(* CODESYS project SPT_XTS.library
   Version: 4.0.0
   Title: SPT XTS
   DefaultNamespace: SPT_XTS
   Placeholder: SPT XTS
   Company: Beckhoff Automation LLC

Project tree, tasks and I/O mapping:
  libraries: SPT Base Types, * (Beckhoff Automation LLC); SPT Event Logger, * (Beckhoff Automation LLC); SPT Utilities, * (Beckhoff Automation LLC); Tc2_Math, * (Beckhoff Automation GmbH); Tc2_MC2, * (Beckhoff Automation GmbH); Tc2_Standard, * (Beckhoff Automation GmbH); Tc2_System, * (Beckhoff Automation GmbH); Tc2_Utilities, * (Beckhoff Automation GmbH); Tc3_EventLogger, * (Beckhoff Automation GmbH); Tc3_JsonXml, * (Beckhoff Automation GmbH); Tc3_McCollisionAvoidance, * (Beckhoff Automation GmbH); Tc3_McCoordinatedMotion, * (Beckhoff Automation GmbH); Tc3_Module, * (Beckhoff Automation GmbH); Tc3_XTS_Utility, * (Beckhoff Automation GmbH); Tc3_PackML_V3, * (Beckhoff Automation GmbH)
  Application Station Reference/
    DUTs/
      data type E_ApplicationStationState
    function block FB_XTS_QueueStation [ST]: CanAcceptMover, CanReleaseMover, Resetting, Execute, GetMovers, MaxNumberOfMovers
    function block FB_XTS_SimpleStation [ST]: Execute, SimulatedProcessTime
  GVLs/
    global variables CONSTANTS
    global variables XTS
  Movers/
    data type E_InitializeState_Mover
    function block FB_XTS_Mover [ST]: CyclicLogic, Disable, Enable, GearInPosCA, JoinGroup, LeaveGroup, MoveAbsoluteCA, MoveRelativeCA, Reset, Stop, Acceleration, Deceleration, Gap, Jerk, Velocity, ActualAcceleration, ActualPosition, ActualPositionModulo, ActualTorque, ActualVelocity, PositionLag, SetAcceleration, SetPosition, SetPositionModulo, SetVelocity, Enabled, InPosition, InSync, Stopped, Axis, IsMoverInPosition, LimitBipolarCurrent, MoverID, Override, Station, Trace, TraceMoveCommand, TraceWriteBoolParameter, TraceWriteParameter, AxisRefLinked, CurrentPart, CurrentPartOID, CurrentTrack, CurrentTrackOID, FB_reinit, Group, Initialize
    interface I_XTS_Mover: Disable, Enable, GearInPosCA, JoinGroup, LeaveGroup, MoveAbsoluteCA, MoveRelativeCA, Reset, Stop, Acceleration, Deceleration, Jerk, Velocity, ActualAcceleration, ActualPosition, ActualPositionModulo, ActualTorque, ActualVelocity, PositionLag, SetAcceleration, SetPosition, SetPositionModulo, SetVelocity, Enabled, InPosition, InSync, Stopped, Axis, IsMoverInPosition, LimitBipolarCurrent, MoverID, Override, Station
    data type ST_GearInPosCAParameters
    data type ST_MoveDynamics
  Parts/
    data type E_InitializeState_Part
    function block FB_XTS_Part [ST]: CyclicLogic, Initialize, ModuleCoEData, Name, ReadyToEnable, Reset
    interface I_XTS_Part: Name, ReadyToEnable
  Project Information/
    function F_GetCompany [ST]
    function F_GetTitle [ST]
    function F_GetVersion [ST]
  Stations/
    data type E_Colors_ARGB
    data type E_InitializeState_Station
    function block FB_XTS_InfoStation [ST]: CyclicLogic, ApplicationStation, Color, GetMover, GetStopPositionOnTrack, MoverQueue, NumberOfStops, StopPositions, GiveMover, StationName, TakeMover, Initialize, IsAQueue, MoverIDsAssigned, ReleaseAllMovers, StationID
    function block FB_XTS_StationBase [ST]: CanAcceptMover, CanReleaseMover, Config, InfoStation, TrackOID, Resetting, Stopping, HMIPermissions, Initialize, GetMovers, GetStopPosition, CyclicLogic, NumberOfAssignedMovers, NumberOfStops, StopPositions
    interface I_XTS_ApplicationStation: CanAcceptMover, CanReleaseMover, Config, InfoStation, Name, TrackOID
    interface I_XTS_InfoStation: ApplicationStation, Color, GetMover, GetStopPositionOnTrack, MoverQueue, NumberOfStops, StopPositions
    interface I_XTS_StationNeighbor: GiveMover, StationName, TakeMover
    data type ST_XTSStationConfig
  Tracks/
    data type E_InitializeState_Track
    function block FB_XTS_Track [ST]: CyclicLogic, GetTrackPositionByPart, IsClosed, Length, Name, Initialize
    interface I_XTS_Track: GetTrackPositionByPart, IsClosed, Length, Name
  Utilities/
    function block FB_MoverQueue [ST]: Clear, Count, Dequeue, Enqueue, FirstMover, LastMover, MoverIDs, Queue
    function block FB_RingBuffer_MCGearInPosCA [ST]: CurrentFB, GetNewFB
    function block FB_RingBuffer_MCMoveAbsoluteCA [ST]: CurrentFB, GetNewFB
    function block FB_RingBuffer_MCMoveRelativeCA [ST]: CurrentFB, GetNewFB
    function block FB_TrackingRegister_Movers [ST]: Check, Clear, NumberCompleted, Reset, Set
    function block FB_TrackingRegister_Stations [ST]: Check, Clear, Complete, NumberCompleted, Reset, Set, StationsToTrack
  Version/
    global variables Global_Version
  XPU/
    DUTs/
      data type E_MoverAssignmentRecoverySource
      data type E_XPUColdStartRecoveryState
      data type E_XPUInitializeState
      data type E_XPUInitializeState_CAGroups
      data type E_XPUInitializeState_Environment
      data type E_XPUInitializeState_InfoStations
      data type E_XPUInitializeState_XPU
      data type E_XTSState
      data type ST_MoverAssignmentData
      data type ST_StationNeighbors
    function block FB_Component_XPU [ST]: CyclicLogic, GetPositionOnTrack, GiveMover, InSimulationMode, CreateEvents, Monitoring, Initialize_CAGroups, Initialize_Environment, Initialize_InfoStations, Initialize_XPU, Initialize, ClearAllEvents, CollectRecoveryData, FindRecoveryCandidates, MoverAssignmentRecovery, ReassignMovers, RestoreBackupData, SetError, SetStationNeighbors, SortMoverBuckets, Trace, ClearMoverAssignments, Disable, Enable, FB_init, MoverAssignmentStorageLocation, PartCoEData, Reset, State, Stations
    interface I_XTS_Xpu: GetPositionOnTrack, GiveMover, InSimulationMode
  00000000-0000-0000-0000-000000000000|LICENSE
  LICENSE
  global variables Parameters_XTS
*)

// Application Station Reference/DUTs/E_ApplicationStationState
{attribute 'qualified_only'}
{attribute 'strict'}
TYPE E_ApplicationStationState : (
		eApplicationStationState_Init		   := 0,
		eApplicationStationState_GetMovers	   := 1,
		eApplicationStationState_InProcess	   := 2,
		eApplicationStationState_ReleaseMovers := 4
	) DWORD;
END_TYPE

// Movers/E_InitializeState_Mover
{attribute 'qualified_only'}
{attribute 'strict'}
TYPE E_InitializeState_Mover : (
		eInitializeStateMover_Check,
		eInitializeStateMover_GetSoftDriveInterfaces,
		eInitializeStateMover_GetSoftDriveInterfaces_Encoder,
		eInitializeStateMover_GetSoftDriveInterfaces_FeedForward,
		eInitializeStateMover_GetSoftDriveInterfaces_Filters,
		eInitializeStateMover_GetSoftDriveInterfaces_Interpolator,
		eInitializeStateMover_GetSoftDriveInterfaces_PositionController,
		eInitializeStateMover_GetSoftDriveInterfaces_VelocityController,
		eInitializeStateMover_ReadTcIOParameters,
		eInitializeStateMover_CheckDriveLinks,
		eInitializeStateMover_ReadNCParameters,
		eInitializeStateMover_Complete,
		eInitializeStateMover_Failed
	);
END_TYPE

// Movers/ST_GearInPosCAParameters
TYPE ST_GearInPosCAParameters :
	STRUCT
		RatioNumerator		: MC_LREAL		   := 1;
		RatioDenumerator	: UINT			   := 1;
		MasterSyncPosition	: MC_LREAL		   := MC_INVALID;
		SlaveSyncPosition	: MC_LREAL		   := MC_INVALID;
		SyncStrategy		: MC_SYNC_STRATEGY := MC_SYNC_STRATEGY.mcSyncStrategyEarly;
		SyncMode			: MC_SYNC_MODE	   := MC_SYNC_MODE.mcSyncModePositive;
		MasterStartDistance : MC_LREAL		   := MC_IGNORE;
		Velocity			: MC_LREAL		   := MC_INVALID;
		Acceleration		: MC_LREAL		   := MC_DEFAULT;
		Deceleration		: MC_LREAL		   := MC_DEFAULT;
		Jerk				: MC_LREAL		   := MC_DEFAULT;
		Gap					: MC_LREAL		   := MC_DEFAULT;
		BufferMode			: MC_BUFFER_MODE   := mcAborting;
		Options				: ST_GearInPosCAOptions;
	END_STRUCT
END_TYPE

// Movers/ST_MoveDynamics
TYPE ST_MoveDynamics :
	STRUCT
		Velocity	 : LREAL := 200;
		Acceleration : LREAL := MC_DEFAULT;
		Deceleration : LREAL := MC_DEFAULT;
		Jerk		 : LREAL := MC_DEFAULT;
	END_STRUCT
END_TYPE

// Parts/E_InitializeState_Part
{attribute 'qualified_only'}
{attribute 'strict'}
TYPE E_InitializeState_Part : (
		eInitializeStatePart_Check,
		eInitializeStatePart_GetModuleInterfaces,
		eInitializeStatePart_GetControlAreaInterfaces,
		eInitializeStatePart_Complete,
		eInitializeStatePart_Failed
	);
END_TYPE

// Stations/E_Colors_ARGB
{attribute 'qualified_only'}
TYPE E_Colors_ARGB : (
		Darkred				 := 16#FF8B0000, //	rgb(139,0,0)
		Brown				 := 16#FFA52A2A, //	rgb(165,42,42)
		Firebrick			 := 16#FFB22222, //	rgb(178,34,34)
		Crimson				 := 16#FFDC143C, //	rgb(220,20,60)
		Red					 := 16#FFFF0000, //	rgb(255,0,0)
		Tomato				 := 16#FFFF6347, //	rgb(255,99,71)
		Coral				 := 16#FFFF7F50, //	rgb(255,127,80)
		Indianred			 := 16#FFCD5C5C, //	rgb(205,92,92)
		Lightcoral			 := 16#FFF08080, //	rgb(240,128,128)
		Darksalmon			 := 16#FFE9967A, //	rgb(233,150,122)
		Salmon				 := 16#FFFA8072, //	rgb(250,128,114)
		Lightsalmon			 := 16#FFFFA07A, //	rgb(255,160,122)
		Orangered			 := 16#FFFF4500, //	rgb(255,69,0)
		Darkorange			 := 16#FFFF8C00, //	rgb(255,140,0)
		Orange				 := 16#FFFFA500, //	rgb(255,165,0)
		Gold				 := 16#FFFFD700, //	rgb(255,215,0)
		Darkgoldenrod		 := 16#FFB8860B, //	rgb(184,134,11)
		Goldenrod			 := 16#FFDAA520, //	rgb(218,165,32)
		Palegoldenrod		 := 16#FFEEE8AA, //	rgb(238,232,170)
		Darkkhaki			 := 16#FFBDB76B, //	rgb(189,183,107)
		Khaki				 := 16#FFF0E68C, //	rgb(240,230,140)
		Olive				 := 16#FF808000, //	rgb(128,128,0)
		Yellow				 := 16#FFFFFF00, //	rgb(255,255,0)
		Yellowgreen			 := 16#FF9ACD32, //	rgb(154,205,50)
		Darkolivegreen		 := 16#FF556B2F, //	rgb(85,107,47)
		Olivedrab			 := 16#FF6B8E23, //	rgb(107,142,35)
		Lawngreen			 := 16#FF7CFC00, //	rgb(124,252,0)
		Chartreuse			 := 16#FF7FFF00, //	rgb(127,255,0)
		Greenyellow			 := 16#FFADFF2F, //	rgb(173,255,47)
		Darkgreen			 := 16#FF006400, //	rgb(0,100,0)
		Green				 := 16#FF008000, //	rgb(0,128,0)
		Forestgreen			 := 16#FF228B22, //	rgb(34,139,34)
		Lime				 := 16#FF00FF00, //	rgb(0,255,0)
		Limegreen			 := 16#FF32CD32, //	rgb(50,205,50)
		Lightgreen			 := 16#FF90EE90, //	rgb(144,238,144)
		Palegreen			 := 16#FF98FB98, //	rgb(152,251,152)
		Darkseagreen		 := 16#FF8FBC8F, //	rgb(143,188,143)
		Mediumspringgreen	 := 16#FF00FA9A, //	rgb(0,250,154)
		Springgreen			 := 16#FF00FF7F, //	rgb(0,255,127)
		Seagreen			 := 16#FF2E8B57, //	rgb(46,139,87)
		Mediumaquamarine	 := 16#FF66CDAA, //	rgb(102,205,170)
		Mediumseagreen		 := 16#FF3CB371, //	rgb(60,179,113)
		Lightseagreen		 := 16#FF20B2AA, //	rgb(32,178,170)
		Darkslategray		 := 16#FF2F4F4F, //	rgb(47,79,79)
		Teal				 := 16#FF008080, //	rgb(0,128,128)
		Darkcyan			 := 16#FF008B8B, //	rgb(0,139,139)
		Aqua				 := 16#FF00FFFF, //	rgb(0,255,255)
		Lightcyan			 := 16#FFE0FFFF, //	rgb(224,255,255)
		Darkturquoise		 := 16#FF00CED1, //	rgb(0,206,209)
		Turquoise			 := 16#FF40E0D0, //	rgb(64,224,208)
		Mediumturquoise		 := 16#FF48D1CC, //	rgb(72,209,204)
		Paleturquoise		 := 16#FFAFEEEE, //	rgb(175,238,238)
		Aquamarine			 := 16#FF7FFFD4, //	rgb(127,255,212)
		Powderblue			 := 16#FFB0E0E6, //	rgb(176,224,230)
		Cadetblue			 := 16#FF5F9EA0, //	rgb(95,158,160)
		Steelblue			 := 16#FF4682B4, //	rgb(70,130,180)
		Cornflowerblue		 := 16#FF6495ED, //	rgb(100,149,237)
		Deepskyblue			 := 16#FF00BFFF, //	rgb(0,191,255)
		Dodgerblue			 := 16#FF1E90FF, //	rgb(30,144,255)
		Lightblue			 := 16#FFADD8E6, //	rgb(173,216,230)
		Skyblue				 := 16#FF87CEEB, //	rgb(135,206,235)
		Lightskyblue		 := 16#FF87CEFA, //	rgb(135,206,250)
		Midnightblue		 := 16#FF191970, //	rgb(25,25,112)
		Navy				 := 16#FF000080, //	rgb(0,0,128)
		Darkblue			 := 16#FF00008B, //	rgb(0,0,139)
		Mediumblue			 := 16#FF0000CD, //	rgb(0,0,205)
		Blue				 := 16#FF0000FF, //	rgb(0,0,255)
		Royalblue			 := 16#FF4169E1, //	rgb(65,105,225)
		Blueviolet			 := 16#FF8A2BE2, //	rgb(138,43,226)
		Indigo				 := 16#FF4B0082, //	rgb(75,0,130)
		Darkslateblue		 := 16#FF483D8B, //	rgb(72,61,139)
		Slateblue			 := 16#FF6A5ACD, //	rgb(106,90,205)
		Mediumslateblue		 := 16#FF7B68EE, //	rgb(123,104,238)
		Mediumpurple		 := 16#FF9370DB, //	rgb(147,112,219)
		Darkmagenta			 := 16#FF8B008B, //	rgb(139,0,139)
		Darkviolet			 := 16#FF9400D3, //	rgb(148,0,211)
		Darkorchid			 := 16#FF9932CC, //	rgb(153,50,204)
		Mediumorchid		 := 16#FFBA55D3, //	rgb(186,85,211)
		Purple				 := 16#FF800080, //	rgb(128,0,128)
		Thistle				 := 16#FFD8BFD8, //	rgb(216,191,216)
		Plum				 := 16#FFDDA0DD, //	rgb(221,160,221)
		Violet				 := 16#FFEE82EE, //	rgb(238,130,238)
		Magenta				 := 16#FFFF00FF, //	rgb(255,0,255)
		Orchid				 := 16#FFDA70D6, //	rgb(218,112,214)
		Mediumvioletred		 := 16#FFC71585, //	rgb(199,21,133)
		Palevioletred		 := 16#FFDB7093, //	rgb(219,112,147)
		Deeppink			 := 16#FFFF1493, //	rgb(255,20,147)
		Hotpink				 := 16#FFFF69B4, //	rgb(255,105,180)
		Lightpink			 := 16#FFFFB6C1, //	rgb(255,182,193)
		Pink				 := 16#FFFFC0CB, //	rgb(255,192,203)
		Antiquewhite		 := 16#FFFAEBD7, //	rgb(250,235,215)
		Beige				 := 16#FFF5F5DC, //	rgb(245,245,220)
		Bisque				 := 16#FFFFE4C4, //	rgb(255,228,196)
		Blanchedalmond		 := 16#FFFFEBCD, //	rgb(255,235,205)
		Wheat				 := 16#FFF5DEB3, //	rgb(245,222,179)
		Cornsilk			 := 16#FFFFF8DC, //	rgb(255,248,220)
		Lemonchiffon		 := 16#FFFFFACD, //	rgb(255,250,205)
		LightGoldenRodYellow := 16#FFFAFAD2, //	rgb(250,250,210)
		LightYellow			 := 16#FFFFFFE0, //	rgb(255,255,224)
		SaddleBrown			 := 16#FF8B4513, //	rgb(139,69,19)
		Sienna				 := 16#FFA0522D, //	rgb(160,82,45)
		Chocolate			 := 16#FFD2691E, //	rgb(210,105,30)
		Peru				 := 16#FFCD853F, //	rgb(205,133,63)
		SandyBrown			 := 16#FFF4A460, //	rgb(244,164,96)
		BurlyWood			 := 16#FFDEB887, //	rgb(222,184,135)
		RosyBrown			 := 16#FFBC8F8F, //	rgb(188,143,143)
		Moccasin			 := 16#FFFFE4B5, //	rgb(255,228,181)
		NavajoWhite			 := 16#FFFFDEAD, //	rgb(255,222,173)
		PeachPuff			 := 16#FFFFDAB9, //	rgb(255,218,185)
		MistyRose			 := 16#FFFFE4E1, //	rgb(255,228,225)
		LavenderBlush		 := 16#FFFFF0F5, //	rgb(255,240,245)
		Linen				 := 16#FFFAF0E6, //	rgb(250,240,230)
		OldLace				 := 16#FFFDF5E6, //	rgb(253,245,230)
		PapayaWhip			 := 16#FFFFEFD5, //	rgb(255,239,213)
		Seashell			 := 16#FFFFF5EE, //	rgb(255,245,238)
		MintCream			 := 16#FFF5FFFA, //	rgb(245,255,250)
		SlateGray			 := 16#FF708090, //	rgb(112,128,144)
		LightSlateGray		 := 16#FF778899, //	rgb(119,136,153)
		LightSteelBlue		 := 16#FFB0C4DE, //	rgb(176,196,222)
		Lavender			 := 16#FFE6E6FA, //	rgb(230,230,250)
		FloralWhite			 := 16#FFFFFAF0, //	rgb(255,250,240)
		AliceBlue			 := 16#FFF0F8FF, //	rgb(240,248,255)
		GhostWhite			 := 16#FFF8F8FF, //	rgb(248,248,255)
		HoneyDew			 := 16#FFF0FFF0, //	rgb(240,255,240)
		Ivory				 := 16#FFFFFFF0, //	rgb(255,255,240)
		Azure				 := 16#FFF0FFFF, //	rgb(240,255,255)
		Snow				 := 16#FFFFFAFA, //	rgb(255,250,250)
		Black				 := 16#FF000000, //	rgb(0,0,0)
		DimGray				 := 16#FF696969, //	rgb(105,105,105)
		Gray				 := 16#FF808080, //	rgb(128,128,128)
		DarkGray			 := 16#FFA9A9A9, //	rgb(169,169,169)
		Silver				 := 16#FFC0C0C0, //	rgb(192,192,192)
		LightGray			 := 16#FFD3D3D3, //	rgb(211,211,211)
		Gainsboro			 := 16#FFDCDCDC, //	rgb(220,220,220)
		WhiteSmoke			 := 16#FFF5F5F5, //	rgb(245,245,245)
		White				 := 16#FFFFFFFF	 //	rgb(255,255,255)
	) UDINT;
END_TYPE

// Stations/E_InitializeState_Station
{attribute 'qualified_only'}
{attribute 'strict'}
TYPE E_InitializeState_Station : (
		eInitializeStateStation_Check,
		eInitializeStateStation_GetPartInfo,
		eInitializeStateStation_GetStopPositions,
		eInitializeStateStation_Complete,
		eInitializeStateStation_Failed
	);
END_TYPE

// Stations/ST_XTSStationConfig
TYPE ST_XTSStationConfig :
	STRUCT
		IsAQueueStation : BOOL; // Can accept movers on cold start recovery (station limits will be ignored!!)
		OverrideGap		: BOOL;
		Gap				: LREAL;
		Dynamics		: ST_MoveDynamics;
	END_STRUCT
END_TYPE

// Tracks/E_InitializeState_Track
{attribute 'qualified_only'}
{attribute 'strict'}
TYPE E_InitializeState_Track : (
		eInitializeStateTrack_Check,
		eInitializeStateTrack_GetPartInfo,
		eInitializeStateTrack_Complete,
		eInitializeStateTrack_Failed
	);
END_TYPE

// XPU/DUTs/E_MoverAssignmentRecoverySource
{attribute 'qualified_only'}
{attribute 'strict'}
TYPE E_MoverAssignmentRecoverySource : (
		eMoverAssignmentRecoverySource_NoBackup	  := 0,
		eMoverAssignmentRecoverySource_NOVRAM	  := 1,
		eMoverAssignmentRecoverySource_Persistent := 2
	);
END_TYPE

// XPU/DUTs/E_XPUColdStartRecoveryState
{attribute 'qualified_only'}
{attribute 'strict'}
TYPE E_XPUColdStartRecoveryState : (
		eXPUColdStartRecoveryState_CheckMover1Config := 0,
		eXPUColdStartRecoveryState_WaitForDriveReady,
		eXPUColdStartRecoveryState_StartMover1Detection,
		eXPUColdStartRecoveryState_WaitForMover1DetectionComplete,
		eXPUColdStartRecoveryState_CheckPersistentDataSource,
		eXPUColdStartRecoveryState_RestorePersistentStationMoverAssignments,
		eXPUColdStartRecoveryState_RestoreNOVRAMStationMoverAssignments,
		eXPUColdStartRecoveryState_LookForRecoveryCandidates,
		eXPUColdStartRecoveryState_ForceMoversOntoCandidates,
		eXPUColdStartRecoveryState_RecoveryComplete
	);
END_TYPE

// XPU/DUTs/E_XPUInitializeState
{attribute 'qualified_only'}
{attribute 'strict'}
TYPE E_XPUInitializeState : (
		eXPUInitializeState_Environment,
		eXPUInitializeState_CAGroups,
		eXPUInitializeState_XPU,
		eXPUInitializeState_InfoStations,
		eXPUInitializeState_Parts,
		eXPUInitializeState_Tracks,
		eXPUInitializeState_Movers,
		eXPUInitializeState_Stations,
		eXPUInitializeState_AttemptMoverRecovery,
		eXPUInitializeState_Complete,
		eXPUInitializeState_Failed
	);
END_TYPE

// XPU/DUTs/E_XPUInitializeState_CAGroups
{attribute 'qualified_only'}
{attribute 'strict'}
TYPE E_XPUInitializeState_CAGroups : (
		eXPUInitializeStateCAGroups_CheckMapping,
		eXPUInitializeStateCAGroups_FindGroupID,
		eXPUInitializeStateCAGroups_CheckGroupInitialized,
		eXPUInitializeStateCAGroups_Complete,
		eXPUInitializeStateCAGroups_Failed
	);
END_TYPE

// XPU/DUTs/E_XPUInitializeState_Environment
{attribute 'qualified_only'}
{attribute 'strict'}
TYPE E_XPUInitializeState_Environment : (
		eXPUInitializeStateEnvironment_Check,
		eXPUInitializeStateEnvironment_InitializeEnvironment,
		eXPUInitializeStateEnvironment_GetXPUCount,
		eXPUInitializeStateEnvironment_GetXPUOIDs,
		eXPUInitializeStateEnvironment_GetInfoServerCounts,
		eXPUInitializeStateEnvironment_GetInfoServerOIDs,
		eXPUInitializeStateEnvironment_GetCAGroupCounts,
		eXPUInitializeStateEnvironment_GetCAGroupOIDs,
		eXPUInitializeStateEnvironment_WaitingForOtherXTS,
		eXPUInitializeStateEnvironment_Cleanup,
		eXPUInitializeStateEnvironment_Complete,
		eXPUInitializeStateEnvironment_Failed
	);
END_TYPE

// XPU/DUTs/E_XPUInitializeState_InfoStations
{attribute 'qualified_only'}
{attribute 'strict'}
TYPE E_XPUInitializeState_InfoStations : (
		eXPUInitializeStateInfoStations_GetInfoServerInterfaces,
		eXPUInitializeStateInfoStations_GetPartOIDs,
		eXPUInitializeStateInfoStations_GetStationCounts,
		eXPUInitializeStateInfoStations_GetStationInterfaces,
		eXPUInitializeStateInfoStations_MatchStationsAgainstParts,
		eXPUInitializeStateInfoStations_Complete,
		eXPUInitializeStateInfoStations_Failed
	);
END_TYPE

// XPU/DUTs/E_XPUInitializeState_XPU
{attribute 'qualified_only'}
{attribute 'strict'}
TYPE E_XPUInitializeState_XPU : (
		eXPUInitializeStateXPU_FindLinkedMover,
		eXPUInitializeStateXPU_FindXPUId,
		eXPUInitializeStateXPU_GetXPUInterface,
		eXPUInitializeStateXPU_GetPartCount,
		eXPUInitializeStateXPU_GetPartInterfaces,
		eXPUInitializeStateXPU_GetTrackCount,
		eXPUInitializeStateXPU_GetTrackInterfaces,
		eXPUInitializeStateXPU_GetMoverCount,
		eXPUInitializeStateXPU_GetMoverInterfaces,
		eXPUInitializeStateXPU_Complete,
		eXPUInitializeStateXPU_Failed
	);
END_TYPE

// XPU/DUTs/E_XTSState
{attribute 'qualified_only'}
{attribute 'strict'}
{attribute 'to_string'}
TYPE E_XTSState : (
		eXTSState_Disabling := 0,
		eXTSState_Disabled	:= 1,
		eXTSState_Enabling	:= 2,
		eXTSState_Enabled	:= 4,
		eXTSState_Error		:= 8,
		eXTSState_Reset		:= 16
	) DWORD;
END_TYPE

// XPU/DUTs/ST_MoverAssignmentData
TYPE ST_MoverAssignmentData :
	STRUCT
		StationID : UDINT;
		MoverIDs  : ARRAY[1..TcIoXtsEnvironmentParameterList.MaxXtsMoversPerXpu] OF UDINT;
	END_STRUCT
END_TYPE

// XPU/DUTs/ST_StationNeighbors
TYPE ST_StationNeighbors :
	STRUCT
		Station			  : I_XTS_StationNeighbor;
		UpstreamStation	  : I_XTS_StationNeighbor;
		DownstreamStation : I_XTS_StationNeighbor;
	END_STRUCT
END_TYPE

// GVLs/CONSTANTS
{attribute 'qualified_only'}
VAR_GLOBAL CONSTANT
	XPU_ALARM_COUNT : UDINT := 18;
END_VAR

// GVLs/XTS
{attribute 'qualified_only'}
VAR_GLOBAL
	Environment				 : Tc3_XTS_Utility.FB_TcIoXtsEnvironment;
	XTSEnvironmentConfig	 : ST_XtsEnvironmentConfiguration := (bEnableInitXPU := TRUE, bEnableInitCaGroup := TRUE, bEnableInitInfoServer := TRUE);
	InitializationInProgress : BOOL;
	InitializationComplete	 : BOOL;
	XPUCount				 : UINT;
	XPUOIDs					 : REFERENCE TO ARRAY[1..TcIoXtsEnvironmentParameterList.MaxXtsProcessingUnits] OF OTCID;
	InfoServerCount			 : UINT;
	InfoServerOIDs			 : REFERENCE TO ARRAY[1..TcIoXtsEnvironmentParameterList.MaxXtsInfoServer] OF OTCID;
	InfoStationCounts		 : ARRAY[1..TcIoXtsEnvironmentParameterList.MaxXtsInfoServer] OF UDINT;
	ipInfoServer			 : ARRAY[1..TcIoXtsEnvironmentParameterList.MaxXtsInfoServer] OF I_TcIoXtsInfoServer;
	ipInfoStations			 : ARRAY[1..TcIoXtsEnvironmentParameterList.MaxXtsInfoServer, 1..TcIoXtsEnvironmentParameterList.MaxXtsInfoStation] OF I_TcIoXtsInfoServerInfoStation;
	CAGroupCount			 : UINT;
	CAGroupOIDs				 : REFERENCE TO ARRAY[1..TcIoXtsEnvironmentParameterList.MaxXtsCaGroup] OF OTCID;
END_VAR

// Version/Global_Version
{attribute 'TcGenerated'}
{attribute 'no-analysis'}
{attribute 'linkalways'}

// This function has been automatically generated from the project information.
VAR_GLOBAL CONSTANT
	{attribute 'const_non_replaced'}
	stLibVersion_SPT_XTS : ST_LibVersion := (iMajor := 4, iMinor := 0, iBuild := 0, iRevision := 0, nFlags := 1, sVersion := '4.0.0');
END_VAR

// Parameters_XTS
{attribute 'qualified_only'}
VAR_GLOBAL CONSTANT
	ALLOW_UNLINKED_MOVER_NC_AXES	   : BOOL		   := FALSE;
	ENABLE_DEBUG_TRACING			   : BOOL		   := FALSE;
	STATIONCOLOR_DEFAULT_GETMOVERS	   : E_Colors_ARGB := E_Colors_ARGB.Yellow;
	STATIONCOLOR_DEFAULT_INPROCESS	   : E_Colors_ARGB := E_Colors_ARGB.Red;
	STATIONCOLOR_DEFAULT_RELEASEMOVERS : E_Colors_ARGB := E_Colors_ARGB.Green;
END_VAR

// Application Station Reference/FB_XTS_QueueStation
FUNCTION_BLOCK FINAL FB_XTS_QueueStation EXTENDS FB_XTS_StationBase
VAR
	_MaxNumberOfMovers : UDINT := TcIoXtsEnvironmentParameterList.MaxXtsMoversPerXpu;
END_VAR

PROPERTY CanAcceptMover : BOOL
GET
CanAcceptMover := NumberOfAssignedMovers < _MaxNumberOfMovers;
END_GET
END_PROPERTY

PROPERTY CanReleaseMover : BOOL
GET
CanReleaseMover := NumberOfAssignedMovers > 0;
END_GET
END_PROPERTY

METHOD PROTECTED Resetting
VAR
	i			 : UDINT;
	ipMovers	 : ARRAY[0..TcIoXtsEnvironmentParameterList.MaxXtsMoversPerXpu] OF I_XTS_Mover;
	StopPosition : LREAL;
END_VAR

VAR_INST
	RecoveryMoveComplete : BOOL; // Initial MoveAbsoluteCA should be in positive direction only--after that we can use ShortestWay
END_VAR
// Need a copy of .Queue so we can index through array
ipMovers := MoverQueue.Queue;
CASE SequenceState OF
	0:
		_Busy := TRUE;
		MoverTracker.Clear();
		SequenceState := SequenceState + 10;

	10:
		// Determine if any movers have been assigned to this station
		IF NumberOfAssignedMovers <> 0 THEN
			SequenceState := 100;
		ELSE
			SequenceState := 1000;
		END_IF

	100:
		MoverTracker.Clear();
		FOR i := 1 TO NumberOfAssignedMovers DO
			IF ipMovers[i] <> 0 THEN
				IF NOT ipMovers[i].Busy THEN
					// Queue stations always command movers to position 1
					StopPosition := StopPositions[1];
					StopPosition := GetStopPosition(StopPosition);
					IF ipMovers[i].MoveAbsoluteCA(StopPosition, TRUE, RecoveryMoveComplete) THEN
						MoverTracker.Set(i);
					END_IF
				END_IF
			END_IF
		END_FOR

		IF MoverTracker.NumberCompleted = NumberOfAssignedMovers THEN
			RecoveryMoveComplete := TRUE;
			SequenceState		 := 1000;
		END_IF

	1000:
		_Busy := FALSE;
		SUPER^.Resetting();
END_CASE
END_METHOD

METHOD PROTECTED Execute
GetMovers();
END_METHOD

METHOD PROTECTED GetMovers : BOOL
VAR
	i			 : UDINT;
	ipMovers	 : ARRAY[0..TcIoXtsEnvironmentParameterList.MaxXtsMoversPerXpu] OF I_XTS_Mover;
	StopPosition : LREAL;
END_VAR
CASE SequenceState OF
	0:
		// Don't combine this with state 20 -- there is a dead scan for method cleanup/returns
		IF CanAcceptMover THEN
			SequenceState := SequenceState + 10;
		END_IF

	10:
		IF ipInfoStation.GetMover() THEN
			// Ask for a new mover		
			SequenceState := SequenceState + 10;
		END_IF

	20:
		// Make sure we don't page fault
		IF MoverQueue.LastMover <> 0 THEN
			// Call new mover to this station--use only stop position 1
			StopPosition := StopPositions[1];
			StopPosition := GetStopPosition(StopPosition);
			IF MoverQueue.LastMover.MoveAbsoluteCA(StopPosition, TRUE, FALSE) THEN
				SequenceState := 0;
			END_IF
		ELSE
			SequenceState := 0;
		END_IF
END_CASE
END_METHOD

PROPERTY MaxNumberOfMovers : UDINT
GET
MaxNumberOfMovers := _MaxNumberOfMovers;
END_GET
SET
_MaxNumberOfMovers := MaxNumberOfMovers;
END_SET
END_PROPERTY

END_FUNCTION_BLOCK

// Stations/FB_XTS_StationBase
FUNCTION_BLOCK ABSTRACT FB_XTS_StationBase EXTENDS FB_PackML_BaseModule IMPLEMENTS I_XTS_ApplicationStation
VAR
	{attribute 'TcInitSymbol'}
	TrackID			  : OTCID;
	ipComponents_Init : ARRAY[1..Parameters_PackML_Base.MAX_NO_OF_COMPONENTS] OF I_ComponentBase := [];
	ipInfoStation	  : I_XTS_InfoStation;
	MoverTracker	  : FB_TrackingRegister_Movers;
	MoverQueue		  : REFERENCE TO FB_MoverQueue;
	StationState	  : E_ApplicationStationState;
	_DisableStation	  : BOOL;
	_StationConfig	  : ST_XTSStationConfig;
END_VAR

PROPERTY CanAcceptMover : BOOL
GET
CanAcceptMover := (StationState = E_ApplicationStationState.eApplicationStationState_GetMovers) OR _DisableStation;
END_GET
END_PROPERTY

PROPERTY CanReleaseMover : BOOL
GET
CanReleaseMover := NumberOfAssignedMovers > 0 AND ((StationState = E_ApplicationStationState.eApplicationStationState_ReleaseMovers) OR _DisableStation);
END_GET
END_PROPERTY

PROPERTY Config : ST_XTSStationConfig
GET
Config := _StationConfig;
END_GET
SET
_StationConfig := Config;
END_SET
END_PROPERTY

PROPERTY InfoStation : I_XTS_InfoStation
SET
ipInfoStation				   := InfoStation;
InfoStation.ApplicationStation := THIS^;
MoverQueue					   REF= ipInfoStation.MoverQueue;
END_SET
END_PROPERTY

PROPERTY TrackOID : OTCID
GET
TrackOID := TrackID;
END_GET
END_PROPERTY

METHOD PROTECTED Resetting
VAR
	i			 : UDINT;
	ipMovers	 : ARRAY[0..TcIoXtsEnvironmentParameterList.MaxXtsMoversPerXpu] OF I_XTS_Mover;
	StopPosition : LREAL;
END_VAR
// Need a copy of .Queue so we can index through array
ipMovers := MoverQueue.Queue;
CASE SequenceState OF
	0:
		_Busy := TRUE;
		MoverTracker.Clear();
		SequenceState := SequenceState + 10;

	10:
		// Determine if any movers have been assigned to this station
		IF NumberOfAssignedMovers <> 0 THEN
			SequenceState := 100;
		ELSE
			SequenceState := 1000;
		END_IF

	100:
		MoverTracker.Clear();
		FOR i := 1 TO NumberOfAssignedMovers DO
			IF ipMovers[i] <> 0 THEN
				IF NOT ipMovers[i].Busy AND_THEN NOT MoverTracker.Check(i) THEN
					StopPosition := StopPositions[NumberOfStops - (i - 1)];
					StopPosition := GetStopPosition(StopPosition);
					IF ipMovers[i].MoveAbsoluteCA(StopPosition, TRUE, TRUE) THEN
						MoverTracker.Set(i);
					END_IF
				END_IF
			END_IF
		END_FOR

		IF MoverTracker.NumberCompleted = NumberOfAssignedMovers THEN
			SequenceState := SequenceState + 10;
		END_IF

	110:
		// Wait for all movers to arrive at their assigned positions
		MoverTracker.Clear();
		FOR i := 1 TO NumberOfAssignedMovers DO
			IF ipMovers[i] <> 0 THEN
				IF NOT ipMovers[i].Busy AND_THEN NOT MoverTracker.Check(i) THEN
					StopPosition := StopPositions[NumberOfStops - (i - 1)];
					StopPosition := GetStopPosition(StopPosition);
					IF ipMovers[i].IsMoverInPosition(StopPosition) THEN
						MoverTracker.Set(i);
					END_IF
				END_IF
			END_IF
		END_FOR

		IF MoverTracker.NumberCompleted = NumberOfAssignedMovers THEN
			SequenceState := 1000;
		END_IF

	1000:
		_Busy := FALSE;
		SUPER^.Resetting();
END_CASE
END_METHOD

METHOD PROTECTED Stopping
VAR
	i			 : UDINT;
	ipMovers	 : ARRAY[0..TcIoXtsEnvironmentParameterList.MaxXtsMoversPerXpu] OF I_XTS_Mover;
	StopPosition : LREAL;
END_VAR
// Need a copy of .Queue so we can index through array
ipMovers := MoverQueue.Queue;
CASE SequenceState OF
	0:
		_Busy := TRUE;
		MoverTracker.Clear();
		SequenceState := SequenceState + 10;

	10:
		// Determine if any movers have been assigned to this station
		IF NumberOfAssignedMovers <> 0 THEN
			SequenceState := 100;
		ELSE
			SequenceState := 1000;
		END_IF

	100:
		// Wait for all movers to arrive at their assigned positions
		MoverTracker.Clear();
		ipMovers := MoverQueue.Queue;
		FOR i := 1 TO NumberOfAssignedMovers DO
			IF ipMovers[i] <> 0 THEN
				IF ipMovers[i].Stopped THEN
					MoverTracker.Set(i);
				END_IF
			END_IF
		END_FOR

		IF MoverTracker.NumberCompleted = NumberOfAssignedMovers THEN
			SequenceState := 1000;
		END_IF

	1000:
		_Busy := FALSE;
		SUPER^.Stopping();
END_CASE
END_METHOD

METHOD PROTECTED HMIPermissions
VAR_INPUT
END_VAR
BlockHMIControl();
END_METHOD

METHOD PROTECTED Initialize : BOOL
VAR
	i : UDINT; // Generic iteration value
END_VAR
Initialize := FALSE;
CASE DescendantSequenceState OF
	0:
		// Define the interfaces to the different subunits (Must take place before SUPER^.initialize call)
		FOR i := 1 TO SPT_BaseTypes.Parameters_PackML_Base.MAX_NO_OF_COMPONENTS DO
			ipComponents[i] := ipComponents_Init[i];
		END_FOR

		_LogModeChanges			:= FALSE;
		_LogStateChanges		:= FALSE;
		DescendantSequenceState := DescendantSequenceState + 10;

	10:
		DescendantSequenceState := DescendantSequenceState + 10;

	20:
		// Copy Mode names
		FOR i := 1 TO 3 DO
			ModeNames[i] := F_PMLUnitModeToString(UDINT_TO_DINT(i));
		END_FOR

		DescendantSequenceState := DescendantSequenceState + 10;

	30:
		// Initialize Recipes 
		DescendantSequenceState := DescendantSequenceState + 10;

	40:
		IF (ipInfoStation <> 0) THEN
			StationState			:= E_ApplicationStationState.eApplicationStationState_GetMovers;
			DescendantSequenceState := DescendantSequenceState + 10;
		END_IF

	50:
		// Call the Super
		IF SUPER^.Initialize() THEN
			DescendantSequenceState := DescendantSequenceState + 10;
		END_IF

	60:
		Initialize := TRUE;
END_CASE
END_METHOD

METHOD PROTECTED GetMovers : BOOL
VAR
	i			 : UDINT;
	ipMovers	 : ARRAY[0..TcIoXtsEnvironmentParameterList.MaxXtsMoversPerXpu] OF I_XTS_Mover;
	StopPosition : LREAL;
END_VAR
CASE SequenceState OF
	0:
		IF (NumberOfAssignedMovers < NumberOfStops) THEN
			SequenceState := SequenceState + 10;
		ELSE
			SequenceState := 40;
		END_IF

	10:
		IF ipInfoStation.GetMover() THEN
			// Ask for a new mover			
			SequenceState := SequenceState + 10;
		END_IF

	20:
		// Make sure we don't page fault
		IF MoverQueue.LastMover <> 0 THEN
			// Call new mover to this station--station positions go front-to-back
			StopPosition := StopPositions[NumberOfStops - (NumberOfAssignedMovers - 1)];
			StopPosition := GetStopPosition(StopPosition);
			IF MoverQueue.LastMover.MoveAbsoluteCA(StopPosition, TRUE, FALSE) THEN
				SequenceState := SequenceState + 10;
			END_IF
		END_IF

	30:
		// Make sure we have the correct number of movers
		IF NumberOfAssignedMovers = NumberOfStops THEN
			SequenceState := SequenceState + 10;
		ELSE
			SequenceState := 10;
		END_IF

	40:
		// Wait for all movers to arrive at their assigned positions
		MoverTracker.Clear();
		ipMovers := MoverQueue.Queue;
		FOR i := 1 TO NumberOfStops DO
			IF ipMovers[i] <> 0 THEN
				IF NOT ipMovers[i].Busy THEN
					StopPosition := StopPositions[NumberOfStops - (i - 1)];
					StopPosition := GetStopPosition(StopPosition);
					IF ipMovers[i].IsMoverInPosition(StopPosition) THEN
						MoverTracker.Set(i);
					END_IF
				END_IF
			END_IF
		END_FOR

		IF MoverTracker.NumberCompleted = NumberOfStops THEN
			SequenceState := SequenceState + 10;
		END_IF

	50:
		SequenceState := 0;
		GetMovers	  := TRUE;
END_CASE
END_METHOD

METHOD PROTECTED GetStopPosition : LREAL
VAR_INPUT
	Position : LREAL;
END_VAR
IF ipInfoStation <> 0 THEN
	GetStopPosition := ipInfoStation.GetStopPositionOnTrack(TrackID, Position);
END_IF
END_METHOD

// This method serves as the entry point for all underlying FB logic

// This method should be called cyclically by descendant function blocks by invoking SUPER^.CyclicLogic().  Alternatively, the contents of this method could be reimplemented entirely in which case a call to this method would not be necessary.
METHOD PUBLIC CyclicLogic
VAR
	i : UDINT;
END_VAR

VAR_INST
	PreviousState : E_ApplicationStationState;
END_VAR
IF ipInfoStation <> 0 THEN
	IF StationState <> PreviousState THEN
		IF NOT _StationConfig.IsAQueueStation THEN
			CASE StationState OF
				E_ApplicationStationState.eApplicationStationState_GetMovers:
					ipInfoStation.Color := Parameters_XTS.STATIONCOLOR_DEFAULT_GETMOVERS;

				E_ApplicationStationState.eApplicationStationState_InProcess:
					ipInfoStation.Color := Parameters_XTS.STATIONCOLOR_DEFAULT_INPROCESS;

				E_ApplicationStationState.eApplicationStationState_ReleaseMovers:
					ipInfoStation.Color := Parameters_XTS.STATIONCOLOR_DEFAULT_RELEASEMOVERS;
			END_CASE
		ELSE
			ipInfoStation.Color := Parameters_XTS.STATIONCOLOR_DEFAULT_RELEASEMOVERS XOR 16#80000000;
		END_IF
	END_IF

	PreviousState := StationState;
END_IF

SUPER^.CyclicLogic();
END_METHOD

PROPERTY NumberOfAssignedMovers : UDINT
GET
IF __ISVALIDREF(MoverQueue) THEN
	NumberOfAssignedMovers := MoverQueue.Count;
END_IF
END_GET
END_PROPERTY

PROPERTY NumberOfStops : UDINT
GET
IF ipInfoStation <> 0 THEN
	NumberOfStops := ipInfoStation.NumberOfStops;
END_IF
END_GET
END_PROPERTY

PROPERTY StopPositions : REFERENCE TO ARRAY[1..TcIoXtsEnvironmentParameterList.MaxXtsStopPositionsPerStation] OF LREAL
GET
IF ipInfoStation <> 0 THEN
	StopPositions REF= ipInfoStation.StopPositions;
END_IF
END_GET
END_PROPERTY

END_FUNCTION_BLOCK

// Stations/I_XTS_ApplicationStation
INTERFACE I_XTS_ApplicationStation

PROPERTY CanAcceptMover : BOOL
GET
END_GET
END_PROPERTY

PROPERTY CanReleaseMover : BOOL
GET
END_GET
END_PROPERTY

PROPERTY Config : ST_XTSStationConfig
GET
END_GET
SET
END_SET
END_PROPERTY

PROPERTY InfoStation : I_XTS_InfoStation
SET
END_SET
END_PROPERTY

PROPERTY Name : STRING
GET
END_GET
END_PROPERTY

PROPERTY TrackOID : OTCID
GET
END_GET
END_PROPERTY

END_INTERFACE

// Stations/I_XTS_InfoStation
INTERFACE I_XTS_InfoStation

PROPERTY ApplicationStation : I_XTS_ApplicationStation
GET
END_GET
SET
END_SET
END_PROPERTY

PROPERTY Color : E_Colors_ARGB
GET
END_GET
SET
END_SET
END_PROPERTY

METHOD GetMover : BOOL
END_METHOD

METHOD GetStopPositionOnTrack : LREAL
VAR_INPUT
	TrackID	 : OTCID;
	Position : LREAL;
END_VAR
END_METHOD

PROPERTY MoverQueue : REFERENCE TO FB_MoverQueue
GET
END_GET
END_PROPERTY

PROPERTY NumberOfStops : UDINT
GET
END_GET
END_PROPERTY

PROPERTY StopPositions : REFERENCE TO ARRAY[1..TcIoXtsEnvironmentParameterList.MaxXtsStopPositionsPerStation] OF LREAL;
GET
END_GET
END_PROPERTY

END_INTERFACE

// Utilities/FB_MoverQueue
//	FIFO Queue for use by stations
FUNCTION_BLOCK FB_MoverQueue
VAR
	MoversInQueue : UDINT := 0;
	ipMovers	  : ARRAY[1..TcIoXtsEnvironmentParameterList.MaxXtsMoversPerXpu] OF I_XTS_Mover;
END_VAR

//	Brute force reset of buffer
METHOD Clear : BOOL
MEMSET(ADR(ipMovers), 0, SIZEOF(ipMovers));
MoversInQueue := 0;
Clear		  := TRUE;
END_METHOD

PROPERTY Count : UDINT
GET
VAR
	i	 : UDINT;
	temp : UDINT;
END_VAR
Count := MoversInQueue;
END_GET
END_PROPERTY

METHOD Dequeue : BOOL
IF MoversInQueue > 0 THEN
	MEMSET(ADR(ipMovers[1]), 0, SIZEOF(ipMovers[1]));
	MoversInQueue := MoversInQueue - 1;
	IF MoversInQueue > 0 THEN
		MEMMOVE(ADR(ipMovers[1]), ADR(ipMovers[2]), SIZEOF(ipMovers[2]) * MoversInQueue);
		MEMSET(ADR(ipMovers[MoversInQueue + 1]), 0, (SIZEOF(ipMovers[1]) * (TcIoXtsEnvironmentParameterList.MaxXtsMoversPerXpu - MoversInQueue)));
	END_IF

	Dequeue := TRUE;
END_IF
END_METHOD

METHOD Enqueue : BOOL
VAR_INPUT
	ipMover : I_XTS_Mover;
END_VAR
IF MoversInQueue < TcIoXtsEnvironmentParameterList.MaxXtsMoversPerXpu THEN
	MoversInQueue			:= MoversInQueue + 1;
	ipMovers[MoversInQueue] := ipMover;
	Enqueue					:= TRUE;
END_IF
END_METHOD

PROPERTY FirstMover : I_XTS_Mover
GET
IF MoversInQueue > 0 THEN
	FirstMover := ipMovers[1];
END_IF
END_GET
END_PROPERTY

PROPERTY LastMover : I_XTS_Mover
GET
IF MoversInQueue > 0 THEN
	LastMover := ipMovers[MoversInQueue];
END_IF
END_GET
END_PROPERTY

PROPERTY MoverIDs : ARRAY[1..TcIoXtsEnvironmentParameterList.MaxXtsMoversPerXpu] OF UDINT
GET
VAR
	i : UDINT;
END_VAR
FOR i := 1 TO MoversInQueue DO
	IF ipMovers[i] <> 0 THEN
		MoverIDs[i] := ipMovers[i].MoverID;
	END_IF
END_FOR
END_GET
END_PROPERTY

PROPERTY Queue : ARRAY[0..TcIoXtsEnvironmentParameterList.MaxXtsMoversPerXpu] OF I_XTS_Mover;
GET
VAR
	i : UDINT;
END_VAR
FOR i := 1 TO MoversInQueue DO
	Queue[i] := ipMovers[i];
END_FOR
END_GET
END_PROPERTY

END_FUNCTION_BLOCK

// Movers/I_XTS_Mover
INTERFACE I_XTS_Mover EXTENDS I_CyclicFB

METHOD PUBLIC Disable : BOOL
END_METHOD

METHOD PUBLIC Enable : BOOL
END_METHOD

METHOD GearInPosCA : BOOL
VAR_INPUT
	Master		  : REFERENCE TO AXIS_REF;
	Parameters	  : ST_GearInPosCAParameters;
	AbortPrevious : BOOL;
END_VAR
END_METHOD

METHOD PUBLIC JoinGroup : BOOL
END_METHOD

METHOD PUBLIC LeaveGroup : BOOL
END_METHOD

METHOD MoveAbsoluteCA : BOOL
VAR_INPUT
	Position	  : LREAL;
	AbortPrevious : BOOL;
	ShortestWay	  : BOOL;
END_VAR
END_METHOD

METHOD PUBLIC MoveRelativeCA : BOOL
VAR_INPUT
	Distance	  : LREAL;
	AbortPrevious : BOOL;
END_VAR
END_METHOD

METHOD Reset : BOOL
END_METHOD

METHOD PUBLIC Stop : BOOL
END_METHOD

PROPERTY Acceleration : LREAL
GET
END_GET
SET
END_SET
END_PROPERTY

PROPERTY Deceleration : LREAL
GET
END_GET
SET
END_SET
END_PROPERTY

PROPERTY Jerk : LREAL
GET
END_GET
SET
END_SET
END_PROPERTY

PROPERTY Velocity : LREAL
GET
END_GET
SET
END_SET
END_PROPERTY

PROPERTY ActualAcceleration : LREAL
GET
END_GET
END_PROPERTY

PROPERTY ActualPosition : LREAL
GET
END_GET
END_PROPERTY

PROPERTY ActualPositionModulo : LREAL
GET
END_GET
END_PROPERTY

PROPERTY ActualTorque : LREAL
GET
END_GET
END_PROPERTY

PROPERTY ActualVelocity : LREAL
GET
END_GET
END_PROPERTY

PROPERTY PositionLag : LREAL
GET
END_GET
END_PROPERTY

PROPERTY SetAcceleration : LREAL
GET
END_GET
END_PROPERTY

PROPERTY SetPosition : LREAL
GET
END_GET
END_PROPERTY

PROPERTY SetPositionModulo : LREAL
GET
END_GET
END_PROPERTY

PROPERTY SetVelocity : LREAL
GET
END_GET
END_PROPERTY

PROPERTY Enabled : BOOL
GET
END_GET
END_PROPERTY

PROPERTY InPosition : BOOL
GET
END_GET
END_PROPERTY

PROPERTY InSync : BOOL
GET
END_GET
END_PROPERTY

PROPERTY Stopped : BOOL
GET
END_GET
END_PROPERTY

PROPERTY Axis : REFERENCE TO AXIS_REF
GET
END_GET
END_PROPERTY

METHOD IsMoverInPosition : BOOL
VAR_INPUT
	Position : LREAL;
END_VAR
END_METHOD

PROPERTY LimitBipolarCurrent : BOOL
GET
END_GET
SET
END_SET
END_PROPERTY

PROPERTY MoverID : UDINT
GET
END_GET
END_PROPERTY

PROPERTY Override : LREAL
GET
END_GET
SET
END_SET
END_PROPERTY

PROPERTY Station : I_XTS_ApplicationStation
SET
END_SET
END_PROPERTY

END_INTERFACE

// Utilities/FB_TrackingRegister_Movers
FUNCTION_BLOCK FB_TrackingRegister_Movers
VAR
	Status : ARRAY[1..TcIoXtsEnvironmentParameterList.MaxXtsMoversPerXpu] OF BOOL;
END_VAR

//This FB is just for ease of tracking what group commands have actually completed

METHOD Check : BOOL
VAR_INPUT
	i : UDINT;
END_VAR
IF (i >= 1) AND (i <= TcIoXtsEnvironmentParameterList.MaxXtsMoversPerXpu) THEN
	Check := Status[i];
END_IF
END_METHOD

METHOD Clear : BOOL
MEMSET(ADR(Status), 0, SIZEOF(Status));
END_METHOD

PROPERTY NumberCompleted : UDINT
GET
VAR
	i : UDINT;
END_VAR
FOR i := 1 TO TcIoXtsEnvironmentParameterList.MaxXtsMoversPerXpu DO
	IF Status[i] THEN
		NumberCompleted := NumberCompleted + 1;
	END_IF
END_FOR
END_GET
END_PROPERTY

METHOD Reset : BOOL
VAR_INPUT
	i : UDINT;
END_VAR
IF (i >= 1) AND (i <= TcIoXtsEnvironmentParameterList.MaxXtsMoversPerXpu) THEN
	Status[i] := FALSE;
END_IF
END_METHOD

METHOD Set : BOOL
VAR_INPUT
	i : UDINT;
END_VAR
IF (i >= 1) AND (i <= TcIoXtsEnvironmentParameterList.MaxXtsMoversPerXpu) THEN
	Status[i] := TRUE;
END_IF
END_METHOD

END_FUNCTION_BLOCK

// Application Station Reference/FB_XTS_SimpleStation
FUNCTION_BLOCK FINAL FB_XTS_SimpleStation EXTENDS FB_XTS_StationBase
VAR
	ProcessSimulationTimer_TON : TON := (PT := T#2S);
	_Pause					   : BOOL;
END_VAR

METHOD PROTECTED Execute
CASE StationState OF
	E_ApplicationStationState.eApplicationStationState_GetMovers:
		IF NOT _DisableStation THEN
			IF GetMovers() THEN
				StationState := E_ApplicationStationState.eApplicationStationState_InProcess;
			END_IF
		END_IF

	E_ApplicationStationState.eApplicationStationState_InProcess:
		ProcessSimulationTimer_TON(IN := NOT _Pause);
		IF ProcessSimulationTimer_TON.Q THEN
			ProcessSimulationTimer_TON(IN := FALSE);
			StationState := E_ApplicationStationState.eApplicationStationState_ReleaseMovers;
		END_IF

	E_ApplicationStationState.eApplicationStationState_ReleaseMovers:
		IF (NumberOfAssignedMovers = 0) THEN
			// Downstream station has accepted all of our movers
			StationState := E_ApplicationStationState.eApplicationStationState_GetMovers;
		END_IF
END_CASE
END_METHOD

PROPERTY SimulatedProcessTime : TIME
GET
SimulatedProcessTime := ProcessSimulationTimer_TON.PT;
END_GET
SET
ProcessSimulationTimer_TON.PT := SimulatedProcessTime;
END_SET
END_PROPERTY

END_FUNCTION_BLOCK

// Movers/FB_XTS_Mover
FUNCTION_BLOCK INTERNAL FB_XTS_Mover EXTENDS FB_CyclicFB IMPLEMENTS I_XTS_Mover
VAR_INPUT
	ipMover : I_TcIoXtsXpuMover;
END_VAR

// Property Backers
VAR
	_Axis			: AXIS_REF;
	_Group			: REFERENCE TO AXES_GROUP_REF;
	_Velocity		: LREAL;
	_Acceleration	: LREAL;
	_Deceleration	: LREAL;
	_Jerk			: LREAL;
	_Gap			: LREAL;
	_AxisParameters : ST_AxisParameterSet;
	ipStation		: I_XTS_ApplicationStation;
	ipCurrentPart	: I_XTS_Part;
	ipCurrentTrack	: I_XTS_Track;
END_VAR

VAR
	ipSoftDrive				   : I_McXtsMoverSoftdrive;
	ipEncoder				   : I_SoftdriveEncoder;
	ipFeedForward			   : I_SoftDriveFeedForward;
	ipFilter1				   : I_SoftDriveFilter1;
	ipFilter2				   : I_SoftDriveFilter2;
	ipInterpolator			   : I_SoftDriveInterpolator;
	ipPositionController	   : I_SoftDrivePositionControl;
	ipVelocityController	   : I_SoftDriveVelocityControl;
	SoftDriveMode		AT %Q* : UINT := 8;
	BipolarCurrentLimit AT %Q* : INT  := 12000;
END_VAR

VAR
	MCPower						: MC_Power;
	MCReset						: MC_Reset;
	RingBuffer_MCMoveRelativeCA : FB_RingBuffer_MCMoveRelativeCA;
	RingBuffer_MCMoveAbsoluteCA : FB_RingBuffer_MCMoveAbsoluteCA;
	RingBuffer_MCGearInPosCA	: FB_RingBuffer_MCGearInPosCA;
	MCGearInPosCA				: POINTER TO MC_GearInPosCA;
	MCMoveRelativeCA			: POINTER TO MC_MoveRelativeCA;
	MCMoveAbsoluteCA			: POINTER TO MC_MoveAbsoluteCA;
	MCHaltCA					: MC_HaltCA;
	MCHalt						: MC_Halt;
	MCAddAxisToGroup			: MC_AddAxisToGroup;
	MCRemoveAxisFromGroup		: MC_RemoveAxisFromGroup;
	MCReadParameterSet			: MC_ReadParameterSet;
	JsonParser					: FB_JsonDomParser;
END_VAR

// Local Variables
VAR
	MasterAxis					 : REFERENCE TO AXIS_REF;
	InitializeState				 : E_InitializeState_Mover;
	BipolarCurrentLimit_Internal : INT := 12000;
	BipolarCurrentLimit_Minimum	 : INT := 0;
	BipolarCurrentLimitRamp		 : FB_SimpleRateLimiter;
	PositionInfo				 : REFERENCE TO ST_PositionInfo;
	EnableCommand				 : BOOL;
END_VAR

METHOD PUBLIC CyclicLogic
IF NOT _InitComplete THEN
	_InitComplete := THIS^.Initialize();
	RETURN;
END_IF

_Axis.ReadStatus();
IF ipMover <> 0 THEN
	PositionInfo REF= ipMover.GetPositionInfo();
END_IF

(* MC_Power *)
MCPower(Axis			:= _Axis,
		Enable			:= EnableCommand,
		Enable_Positive := TRUE,
		Enable_Negative := TRUE);

IF MCPower.Error THEN
	_Error	 := TRUE;
	_ErrorID := MCPower.ErrorID;
END_IF

(* MC_Reset *)
MCReset(Axis := _Axis);
IF NOT MCReset.Busy THEN
	IF MCReset.Error THEN
		IF Parameters_XTS.ENABLE_DEBUG_TRACING THEN
			Trace('MCReset Error');
		END_IF

		_Error	 := TRUE;
		_ErrorID := MCReset.ErrorID;
	ELSIF MCReset.Done THEN
		IF Parameters_XTS.ENABLE_DEBUG_TRACING THEN
			Trace('MCReset Command Succeeded');
		END_IF
	END_IF

	MCReset(Axis := _Axis, Execute := FALSE);
END_IF

(* MC_MoveRelativeCA *)
RingBuffer_MCMoveRelativeCA(Axis := _Axis);
IF (MCMoveRelativeCA <> 0) AND_THEN NOT MCMoveRelativeCA^.Busy THEN
	IF MCMoveRelativeCA^.Error THEN
		IF Parameters_XTS.ENABLE_DEBUG_TRACING THEN
			Trace('MCMoveRelativeCA Error');
		END_IF

		_Error	 := TRUE;
		_ErrorID := MCMoveRelativeCA^.ErrorID;
	ELSIF MCMoveRelativeCA^.CommandAborted THEN
		IF Parameters_XTS.ENABLE_DEBUG_TRACING THEN
			Trace('MCMoveRelativeCA Command Aborted');
		END_IF
	ELSIF MCMoveAbsoluteCA^.Done THEN
		IF Parameters_XTS.ENABLE_DEBUG_TRACING THEN
			Trace('MCMoveRelativeCA Command Succeeded');
		END_IF
	END_IF

	MCMoveRelativeCA^(Axis := _Axis, Execute := FALSE);
END_IF

(* MC_MoveAbsoluteCA *)
RingBuffer_MCMoveAbsoluteCA(Axis := _Axis);
IF (MCMoveAbsoluteCA <> 0) AND_THEN NOT MCMoveAbsoluteCA^.Busy THEN
	IF MCMoveAbsoluteCA^.Error THEN
		IF Parameters_XTS.ENABLE_DEBUG_TRACING THEN
			Trace('MCMoveAbsoluteCA Error');
		END_IF

		_Error	 := TRUE;
		_ErrorID := MCMoveAbsoluteCA^.ErrorID;
	ELSIF MCMoveAbsoluteCA^.CommandAborted THEN
		IF Parameters_XTS.ENABLE_DEBUG_TRACING THEN
			Trace('MCMoveAbsoluteCA Command Aborted');
		END_IF
	ELSIF MCMoveAbsoluteCA^.Done THEN
		IF Parameters_XTS.ENABLE_DEBUG_TRACING THEN
			Trace('MCMoveAbsoluteCA Command Succeeded');
		END_IF
	END_IF

	MCMoveAbsoluteCA^(Axis := _Axis, Execute := FALSE);
END_IF

(* MC_GearInPoCA *)
RingBuffer_MCGearInPosCA(Master := MasterAxis, Slave := _Axis);
IF (MCGearInPosCA <> 0) AND_THEN NOT MCGearInPosCA^.Busy THEN
	IF MCGearInPosCA^.Error THEN
		IF Parameters_XTS.ENABLE_DEBUG_TRACING THEN
			Trace('MCGearInPosCA Error');
		END_IF

		_Error	 := TRUE;
		_ErrorID := MCGearInPosCA^.ErrorID;
	ELSIF MCGearInPosCA^.CommandAborted THEN
		IF Parameters_XTS.ENABLE_DEBUG_TRACING THEN
			Trace('MCGearInPosCA Command Aborted');
		END_IF
	ELSIF MCGearInPosCA^.InSync THEN
		IF Parameters_XTS.ENABLE_DEBUG_TRACING THEN
			Trace('MCGearInPosCA Command Succeeded');
		END_IF
	END_IF

	MCGearInPosCA^(Master := MasterAxis, Slave := _Axis, Execute := FALSE);
END_IF

(* MC_MCHaltCA *)
MCHaltCA(Axis := _Axis, Deceleration := _Deceleration);
IF NOT MCHaltCA.Busy THEN
	IF MCHaltCA.Error THEN
		IF Parameters_XTS.ENABLE_DEBUG_TRACING THEN
			Trace('MCHaltCA Error');
		END_IF

		_Error	 := TRUE;
		_ErrorID := MCHaltCA.ErrorID;
	ELSIF MCHaltCA.CommandAborted THEN
		IF Parameters_XTS.ENABLE_DEBUG_TRACING THEN
			Trace('MCHaltCA Command Aborted');
		END_IF
	ELSIF MCHaltCA.Done THEN
		IF Parameters_XTS.ENABLE_DEBUG_TRACING THEN
			Trace('MCHaltCA Command Succeeded');
		END_IF
	END_IF

	MCHaltCA(Axis := _Axis, Execute := FALSE);
END_IF

(* MC_MCHalt *)
MCHalt(Axis := _Axis, Deceleration := _Deceleration);
IF NOT MCHalt.Busy THEN
	IF MCHalt.Error THEN
		IF Parameters_XTS.ENABLE_DEBUG_TRACING THEN
			Trace('MCHalt Error');
		END_IF

		_Error	 := TRUE;
		_ErrorID := MCHalt.ErrorID;
	ELSIF MCHalt.CommandAborted THEN
		IF Parameters_XTS.ENABLE_DEBUG_TRACING THEN
			Trace('MCHalt Command Aborted');
		END_IF
	ELSIF MCHalt.Done THEN
		IF Parameters_XTS.ENABLE_DEBUG_TRACING THEN
			Trace('MCHalt Command Succeeded');
		END_IF
	END_IF

	MCHalt(Axis := _Axis, Execute := FALSE);
END_IF

(* Group Functions *)
IF __ISVALIDREF(_Group) THEN
	MCAddAxisToGroup(AxesGroup := _Group, Axis := _Axis, IdentInGroup := UDINT_TO_IDENTINGROUP(_Axis.NcToPlc.AxisId));
	IF NOT MCAddAxisToGroup.Busy THEN
		IF MCAddAxisToGroup.Error THEN
			IF Parameters_XTS.ENABLE_DEBUG_TRACING THEN
				Trace('MCAddAxisToGroup Error');
			END_IF

			_Error	 := TRUE;
			_ErrorID := MCAddAxisToGroup.ErrorID;
		ELSIF MCAddAxisToGroup.Done THEN
			IF Parameters_XTS.ENABLE_DEBUG_TRACING THEN
				Trace('MCAddAxisToGroup Command Succeeded');
			END_IF
		END_IF

		MCAddAxisToGroup(AxesGroup := _Group, Axis := _Axis, Execute := FALSE);
	END_IF

	MCRemoveAxisFromGroup(AxesGroup := _Group, IdentInGroup := UDINT_TO_IDENTINGROUP(_Axis.NcToPlc.AxisId));
	IF NOT MCRemoveAxisFromGroup.Busy THEN
		IF MCRemoveAxisFromGroup.Error THEN
			IF Parameters_XTS.ENABLE_DEBUG_TRACING THEN
				Trace('MCRemoveAxisFromGroup Error');
			END_IF

			_Error	 := TRUE;
			_ErrorID := MCRemoveAxisFromGroup.ErrorID;
		ELSIF MCRemoveAxisFromGroup.Done THEN
			IF Parameters_XTS.ENABLE_DEBUG_TRACING THEN
				Trace('MCRemoveAxisFromGroup Command Succeeded');
			END_IF
		END_IF

		MCRemoveAxisFromGroup(AxesGroup := _Group, IdentInGroup := UDINT_TO_IDENTINGROUP(_Axis.NcToPlc.AxisId), Execute := FALSE);
	END_IF
END_IF

IF _Axis.Status.Error THEN
	_Error	 := TRUE;
	_ErrorID := _Axis.Status.ErrorID;
END_IF

BipolarCurrentLimitRamp(Enable		  := TRUE,
						TargetValue	  := INT_TO_LREAL(BipolarCurrentLimit_Internal),
						Minimum		  := 0,
						Maximum		  := 12000.0,
						Rate_Increase := 12000.0,
						Rate_Decrease := 120000.0);

BipolarCurrentLimit := LREAL_TO_INT(BipolarCurrentLimitRamp.Y);
_Busy				:= (MCReset.Busy OR MCHalt.Busy OR MCHaltCA.Busy OR MCAddAxisToGroup.Busy OR MCRemoveAxisFromGroup.Busy OR MCReadParameterSet.Busy) OR ((MCMoveRelativeCA <> 0) AND_THEN MCMoveRelativeCA^.Busy) OR ((MCMoveAbsoluteCA <> 0) AND_THEN MCMoveAbsoluteCA^.Busy);
END_METHOD

METHOD Disable : BOOL
IF EnableCommand THEN
	EnableCommand := FALSE;
	IF Parameters_XTS.ENABLE_DEBUG_TRACING THEN
		Trace('Disable Command Called');
	END_IF
ELSE
	Disable := NOT MCPower.Status;
END_IF
END_METHOD

METHOD Enable : BOOL
IF NOT _Error THEN
	IF NOT EnableCommand THEN
		EnableCommand := TRUE;
		IF Parameters_XTS.ENABLE_DEBUG_TRACING THEN
			Trace('Enable Command Called');
		END_IF
	ELSE
		Enable := MCPower.Status;
	END_IF
END_IF
END_METHOD

METHOD GearInPosCA : BOOL
VAR_INPUT
	Master		  : REFERENCE TO AXIS_REF;
	Parameters	  : ST_GearInPosCAParameters;
	AbortPrevious : BOOL;
END_VAR
IF _Error THEN
	RETURN;
ELSE
	IF (_Busy AND NOT AbortPrevious) THEN
		RETURN;
	END_IF
END_IF

MasterAxis REF= Master;
IF NOT __ISVALIDREF(MasterAxis) THEN
	RETURN;
END_IF

MCGearInPosCA := RingBuffer_MCGearInPosCA.GetNewFB();
MCGearInPosCA^(Master			   := MasterAxis,
			   Slave			   := _Axis,
			   Execute			   := TRUE,
			   RatioNumerator	   := Parameters.RatioNumerator,
			   RatioDenumerator	   := Parameters.RatioDenumerator,
			   MasterSyncPosition  := Parameters.MasterSyncPosition,
			   SlaveSyncPosition   := Parameters.SlaveSyncPosition,
			   SyncStrategy		   := Parameters.SyncStrategy,
			   SyncMode			   := Parameters.SyncMode,
			   MasterStartDistance := Parameters.MasterStartDistance,
			   Velocity			   := Parameters.Velocity,
			   Acceleration		   := Parameters.Acceleration,
			   Deceleration		   := Parameters.Deceleration,
			   Jerk				   := Parameters.Jerk,
			   Gap				   := Parameters.Gap,
			   Options			   := Parameters.Options);

IF Parameters_XTS.ENABLE_DEBUG_TRACING THEN
	Trace('GearInPosCA');
END_IF

_Busy		:= TRUE;
GearInPosCA := TRUE;
END_METHOD

METHOD PUBLIC JoinGroup : BOOL
IF __ISVALIDREF(_Group) AND NOT _Busy AND NOT _Error THEN
	IF Parameters_XTS.ENABLE_DEBUG_TRACING THEN
		Trace('Join Group Command Called');
	END_IF

	MCAddAxisToGroup(AxesGroup	  := _Group,
					 Axis		  := _Axis,
					 IdentInGroup := UDINT_TO_IDENTINGROUP(_Axis.NcToPlc.AxisId),
					 Execute	  := TRUE);

	_Busy	  := TRUE;
	JoinGroup := TRUE;
END_IF
END_METHOD

METHOD PUBLIC LeaveGroup : BOOL
IF __ISVALIDREF(_Group) AND NOT _Busy AND NOT _Error THEN
	IF Parameters_XTS.ENABLE_DEBUG_TRACING THEN
		Trace('Leave Group Command Called');
	END_IF

	MCRemoveAxisFromGroup(AxesGroup := _Group, Execute := TRUE);
	_Busy	   := TRUE;
	LeaveGroup := TRUE;
END_IF
END_METHOD

//	Absolute positioning move with collision avoidance.	Allows for interruption by toggling between fbMC..A and fbMC..B
METHOD PUBLIC MoveAbsoluteCA : BOOL
VAR_INPUT
	Position	  : LREAL;
	AbortPrevious : BOOL;
	ShortestWay	  : BOOL;
END_VAR

VAR
	StationConfig : ST_XTSStationConfig;
	MoveDynamics  : ST_MoveDynamics; // Could be station-specific
END_VAR
IF _Error THEN
	RETURN;
ELSE
	IF (_Busy AND NOT AbortPrevious) THEN
		RETURN;
	END_IF
END_IF

MCMoveAbsoluteCA := RingBuffer_MCMoveAbsoluteCA.GetNewFB();

// Use station-specific dynamics
IF ipStation <> 0 THEN
	StationConfig := ipStation.Config;
	MoveDynamics  := StationConfig.Dynamics;
	IF StationConfig.OverrideGap THEN
		// Station has a specified gapping other than default
		MCMoveAbsoluteCA^.Gap := StationConfig.Gap;
	ELSE
		MCMoveAbsoluteCA^.Gap := MC_DEFAULT;
	END_IF
ELSE
	MoveDynamics.Velocity	  := _Velocity;
	MoveDynamics.Acceleration := _Acceleration;
	MoveDynamics.Deceleration := _Deceleration;
	MoveDynamics.Jerk		  := _Jerk;
	MCMoveAbsoluteCA^.Gap	  := MC_DEFAULT;
END_IF

IF ShortestWay THEN
	MCMoveAbsoluteCA^.Direction := Tc3_Mc3Definitions.MC_DIRECTION.mcDirectionShortestWay;
ELSE
	MCMoveAbsoluteCA^.Direction := Tc3_Mc3Definitions.MC_DIRECTION.mcDirectionPositive;
END_IF

MCMoveAbsoluteCA^(Axis		   := _Axis,
				  Execute	   := TRUE,
				  Position	   := Position,
				  Velocity	   := MoveDynamics.Velocity,
				  Acceleration := MoveDynamics.Acceleration,
				  Deceleration := MoveDynamics.Deceleration,
				  Jerk		   := MoveDynamics.Jerk);

IF Parameters_XTS.ENABLE_DEBUG_TRACING THEN
	TraceMoveCommand('MoveAbsoluteCA',
					 Position,
					 MoveDynamics.Velocity,
					 MoveDynamics.Acceleration,
					 MoveDynamics.Deceleration,
					 MCMoveAbsoluteCA^.Gap);
END_IF

_Busy		   := TRUE;
MoveAbsoluteCA := TRUE;
END_METHOD

// Relative positioning move with collision avoidance
METHOD PUBLIC MoveRelativeCA : BOOL
VAR_INPUT
	Distance	  : LREAL;
	AbortPrevious : BOOL;
END_VAR

VAR
	StationConfig : ST_XTSStationConfig;
	MoveDynamics  : ST_MoveDynamics; // Could be station-specific
END_VAR
IF _Error THEN
	RETURN;
ELSE
	IF (_Busy AND NOT AbortPrevious) THEN
		RETURN;
	END_IF
END_IF

MCMoveRelativeCA := RingBuffer_MCMoveRelativeCA.GetNewFB();

// Use station-specific dynamics
IF ipStation <> 0 THEN
	StationConfig := ipStation.Config;
	MoveDynamics  := StationConfig.Dynamics;
	IF StationConfig.OverrideGap THEN
		// Station has a specified gapping other than default
		MCMoveRelativeCA^.Gap := StationConfig.Gap;
	ELSE
		MCMoveRelativeCA^.Gap := MC_DEFAULT;
	END_IF
ELSE
	MoveDynamics.Velocity	  := _Velocity;
	MoveDynamics.Acceleration := _Acceleration;
	MoveDynamics.Deceleration := _Deceleration;
	MoveDynamics.Jerk		  := _Jerk;
	MCMoveRelativeCA^.Gap	  := MC_DEFAULT;
END_IF

MCMoveRelativeCA^(Axis		   := _Axis,
				  Execute	   := TRUE,
				  Distance	   := Distance,
				  Velocity	   := MoveDynamics.Velocity,
				  Acceleration := MoveDynamics.Acceleration,
				  Deceleration := MoveDynamics.Deceleration,
				  Jerk		   := MoveDynamics.Jerk);

IF Parameters_XTS.ENABLE_DEBUG_TRACING THEN
	TraceMoveCommand('MoveRelativeCA',
					 Distance,
					 MoveDynamics.Velocity,
					 MoveDynamics.Acceleration,
					 MoveDynamics.Deceleration,
					 MCMoveRelativeCA^.Gap);
END_IF

_Busy		   := TRUE;
MoveRelativeCA := TRUE;
END_METHOD

METHOD Reset : BOOL
IF _Busy THEN
	RETURN;
END_IF

MCReset(Axis := _Axis, Execute := TRUE);
IF MCMoveRelativeCA <> 0 THEN
	IF MCMoveRelativeCA^.Error THEN
		MCMoveRelativeCA^(Axis := _Axis, Execute := FALSE);
	END_IF
END_IF

IF MCMoveAbsoluteCA <> 0 THEN
	IF MCMoveAbsoluteCA^.Error THEN
		MCMoveAbsoluteCA^(Axis := _Axis, Execute := FALSE);
	END_IF
END_IF

IF MCHaltCA.Error THEN
	MCHaltCA(Axis := _Axis, Execute := FALSE);
END_IF

IF MCHalt.Error THEN
	MCHalt(Axis := _Axis, Execute := FALSE);
END_IF

IF __ISVALIDREF(_Group) THEN
	IF MCAddAxisToGroup.Error THEN
		MCAddAxisToGroup(Axis := _Axis, AxesGroup := _Group, Execute := FALSE);
	END_IF

	IF MCRemoveAxisFromGroup.Error THEN
		MCRemoveAxisFromGroup(AxesGroup := _Group, Execute := FALSE);
	END_IF
END_IF

IF MCReadParameterSet.Error THEN
	MCReadParameterSet(Axis := _Axis, Parameter := _AxisParameters, Execute := FALSE);
END_IF

IF Parameters_XTS.ENABLE_DEBUG_TRACING THEN
	Trace('Reset Command Called');
END_IF

_Error	 := FALSE;
_ErrorID := 0;
Reset	 := TRUE;
END_METHOD

// Allow halt commands regardless of other commands being active (do not evaluate _Busy)
METHOD Stop : BOOL
IF _Error THEN
	RETURN;
ELSE
	IF _Axis.Status.ExtSetPointGenEnabled THEN
		// We are in a group so use MCHaltCA
		IF NOT MCHaltCA.Busy THEN
			_Busy := TRUE;
			IF Parameters_XTS.ENABLE_DEBUG_TRACING THEN
				TraceMoveCommand('Halt Command Called - Using MCHaltCA',
								 0,
								 0,
								 _Acceleration,
								 _Deceleration,
								 0);
			END_IF

			MCHaltCA(Axis		  := _Axis,
					 Execute	  := TRUE,
					 Deceleration := _Deceleration,
					 Jerk		  := _Jerk);

			Stop := TRUE;
		END_IF
	ELSE
		// Use standard MCHalt if axis is not in a group (MCHaltCA will fault)
		IF NOT MCHalt.Busy THEN
			_Busy := TRUE;
			IF Parameters_XTS.ENABLE_DEBUG_TRACING THEN
				TraceMoveCommand('Halt Command Called - Using MCHalt',
								 0,
								 0,
								 _Acceleration,
								 _Deceleration,
								 0);
			END_IF

			MCHalt(Axis			:= _Axis,
				   Execute		:= TRUE,
				   Deceleration := _Deceleration,
				   Jerk			:= _Jerk);

			Stop := TRUE;
		END_IF
	END_IF
END_IF
END_METHOD

PROPERTY Acceleration : LREAL
GET
Acceleration := _Acceleration;
END_GET
SET
_Acceleration := Acceleration;
END_SET
END_PROPERTY

PROPERTY Deceleration : LREAL
GET
Deceleration := _Deceleration;
END_GET
SET
_Deceleration := Deceleration;
END_SET
END_PROPERTY

PROPERTY Gap : LREAL
GET
Gap := _Gap;
END_GET
SET
_Gap := Gap;
END_SET
END_PROPERTY

PROPERTY Jerk : LREAL
GET
Jerk := _Jerk;
END_GET
SET
_Jerk := Jerk;
END_SET
END_PROPERTY

PROPERTY Velocity : LREAL
GET
Velocity := _Velocity;
END_GET
SET
_Velocity := Velocity;
END_SET
END_PROPERTY

PROPERTY ActualAcceleration : LREAL
GET
ActualAcceleration := _Axis.NcToPlc.ActAcc;
END_GET
END_PROPERTY

PROPERTY ActualPosition : LREAL
GET
ActualPosition := _Axis.NcToPlc.ActPos;
END_GET
END_PROPERTY

PROPERTY ActualPositionModulo : LREAL
GET
ActualPositionModulo := _Axis.NcToPlc.ModuloActPos;
END_GET
END_PROPERTY

PROPERTY ActualTorque : LREAL
GET
ActualTorque := _Axis.NcToPlc.ActTorque;
END_GET
END_PROPERTY

PROPERTY ActualVelocity : LREAL
GET
ActualVelocity := _Axis.NcToPlc.ActVelo;
END_GET
END_PROPERTY

PROPERTY PositionLag : LREAL
GET
PositionLag := _Axis.NcToPlc.PosDiff;
END_GET
END_PROPERTY

PROPERTY SetAcceleration : LREAL
GET
SetAcceleration := _Axis.NcToPlc.SetAcc;
END_GET
END_PROPERTY

PROPERTY SetPosition : LREAL
GET
SetPosition := _Axis.NcToPlc.SetPos;
END_GET
END_PROPERTY

PROPERTY SetPositionModulo : LREAL
GET
SetPositionModulo := PositionInfo.fTrackPosition;
END_GET
END_PROPERTY

PROPERTY SetVelocity : LREAL
GET
SetVelocity := Axis.NcToPlc.SetVelo;
END_GET
END_PROPERTY

PROPERTY Enabled : BOOL
GET
Enabled := MCPower.Status;
END_GET
END_PROPERTY

PROPERTY InPosition : BOOL
GET
InPosition := _Axis.Status.InTargetPosition;
END_GET
END_PROPERTY

PROPERTY InSync : BOOL
GET
IF MCGearInPosCA <> 0 THEN
	InSync := MCGearInPosCA^.InSync;
END_IF
END_GET
END_PROPERTY

PROPERTY Stopped : BOOL
GET
Stopped := _Axis.Status.NotMoving OR _Axis.Status.Disabled;
END_GET
END_PROPERTY

PROPERTY Axis : REFERENCE TO AXIS_REF
GET
Axis REF= _Axis;
END_GET
END_PROPERTY

METHOD IsMoverInPosition : BOOL
VAR_INPUT
	Position : LREAL;
END_VAR

VAR
	CurrentPosition	  : LREAL;
	PositionTolerance : LREAL;
	MinPosition		  : LREAL;
	MaxPosition		  : LREAL;
END_VAR
IF NOT (ipCurrentTrack <> 0) THEN
	RETURN;
END_IF

CurrentPosition	  := PositionInfo.fTrackPosition;
PositionTolerance := _AxisParameters.fTargetPosControlRange;
IF ipCurrentTrack.IsClosed THEN
	MinPosition := MODABS((Position - PositionTolerance), ipCurrentTrack.Length);
	MaxPosition := MODABS((Position + PositionTolerance), ipCurrentTrack.Length);
	IF (MinPosition + PositionTolerance) > ipCurrentTrack.Length THEN
		// Test range straddles zero
		IsMoverInPosition := (CurrentPosition >= MinPosition) OR (CurrentPosition <= MaxPosition);
	ELSE
		IF MaxPosition = 0 THEN
			// Max is right on the modulo rollover point
			MaxPosition := ipCurrentTrack.Length;
		END_IF

		IsMoverInPosition := (CurrentPosition >= MinPosition) AND (CurrentPosition <= MaxPosition);
	END_IF
ELSE
	IF (Position - PositionTolerance) < 0 THEN
		MinPosition := 0;
	ELSE
		MinPosition := Position - PositionTolerance;
	END_IF

	IF (Position + PositionTolerance) > ipCurrentTrack.Length THEN
		MaxPosition := ipCurrentTrack.Length;
	ELSE
		MaxPosition := Position + PositionTolerance;
	END_IF

	IsMoverInPosition := (CurrentPosition >= MinPosition) AND (CurrentPosition <= MaxPosition);
END_IF
END_METHOD

PROPERTY LimitBipolarCurrent : BOOL
GET
LimitBipolarCurrent := (BipolarCurrentLimit_Internal = BipolarCurrentLimit_Minimum);
END_GET
SET
IF LimitBipolarCurrent THEN
	BipolarCurrentLimit_Internal := BipolarCurrentLimit_Minimum;
ELSE
	BipolarCurrentLimit_Internal := 12000;
END_IF
END_SET
END_PROPERTY

PROPERTY MoverID : UDINT
GET
MoverID := _Axis.NcToPlc.AxisId;
END_GET
END_PROPERTY

PROPERTY Override : LREAL
GET
Override := MCPower.Override;
END_GET
SET
IF Override >= 0 AND Override <= 100 THEN
	MCPower.Override := Override;
END_IF
END_SET
END_PROPERTY

PROPERTY Station : I_XTS_ApplicationStation
SET
IF Parameters_XTS.ENABLE_DEBUG_TRACING THEN
	Trace(CONCAT('Mover ', CONCAT(TO_STRING(MoverID), CONCAT(' is now assigned to ', Station.Name))));
END_IF

ipStation := Station;
END_SET
END_PROPERTY

METHOD PRIVATE Trace
VAR_INPUT
	Message : T_MaxString;
END_VAR

VAR
	Document	  : SJsonValue;
	XTSJsonObject : SJsonValue;
	TempString	  : T_MaxString;
	JsonAttribute : T_MaxString;
END_VAR
{analysis -62}
Document := JsonParser.NewDocument();
JsonParser.AddObjectMember(Document, 'Mover');
XTSJsonObject := JsonParser.FindMember(Document, 'Mover');
JsonParser.AddUintMember(XTSJsonObject, 'AxisID', Axis.NcToPlc.AxisId);
IF ipMover <> 0 THEN
	TempString := ipMover.GetObjectName();
	JsonParser.AddStringMember(XTSJsonObject, 'Name', TempString);
END_IF

IF ipCurrentTrack <> 0 THEN
	TempString := ipCurrentTrack.Name;
	JsonParser.AddStringMember(XTSJsonObject, 'Track', TempString);
ELSE
	JsonParser.AddStringMember(XTSJsonObject, 'Track', 'null');
END_IF

IF ipCurrentPart <> 0 THEN
	TempString := ipCurrentPart.Name;
	JsonParser.AddStringMember(XTSJsonObject, 'Part', TempString);
ELSE
	JsonParser.AddStringMember(XTSJsonObject, 'Part', 'null');
END_IF

IF __ISVALIDREF(PositionInfo) THEN
	TempString := LREAL_TO_FMTSTR(PositionInfo.fTrackPosition, 3, TRUE);
	JsonParser.AddStringMember(XTSJsonObject, 'ActPos', TempString);
ELSE
	TempString := LREAL_TO_FMTSTR(_Axis.NcToPlc.ModuloActPos, 3, TRUE);
	JsonParser.AddStringMember(XTSJsonObject, 'ActPos', TempString);
END_IF

TempString := LREAL_TO_FMTSTR(_Axis.NcToPlc.ActVelo, 3, TRUE);
JsonParser.AddStringMember(XTSJsonObject, 'ActVel', TempString);
TempString := LREAL_TO_FMTSTR(_Axis.NcToPlc.PosDiff, 3, TRUE);
JsonParser.AddStringMember(XTSJsonObject, 'PosLag', TempString);
TraceWithJson(Message, JsonParser.GetJson(Document));
END_METHOD

METHOD PRIVATE TraceMoveCommand
VAR_INPUT
	MoveType	 : T_MaxString;
	Position	 : LREAL;
	Velocity	 : LREAL;
	Acceleration : LREAL;
	Deceleration : LREAL;
	Gap			 : LREAL;
END_VAR

VAR
	Message		  : T_MaxString;
	Document	  : SJsonValue;
	XTSJsonObject : SJsonValue;
	TempString	  : T_MaxString;
	JsonAttribute : T_MaxString;
END_VAR
{analysis -62}
Document := JsonParser.NewDocument();
JsonParser.AddObjectMember(Document, 'Mover');
XTSJsonObject := JsonParser.FindMember(Document, 'Mover');
JsonParser.AddUintMember(XTSJsonObject, 'AxisID', Axis.NcToPlc.AxisId);
IF ipMover <> 0 THEN
	TempString := ipMover.GetObjectName();
	JsonParser.AddStringMember(XTSJsonObject, 'Name', TempString);
END_IF

IF ipCurrentTrack <> 0 THEN
	TempString := ipCurrentTrack.Name;
	JsonParser.AddStringMember(XTSJsonObject, 'Track', TempString);
ELSE
	JsonParser.AddStringMember(XTSJsonObject, 'Track', 'null');
END_IF

IF ipCurrentPart <> 0 THEN
	TempString := ipCurrentPart.Name;
	JsonParser.AddStringMember(XTSJsonObject, 'Part', TempString);
ELSE
	JsonParser.AddStringMember(XTSJsonObject, 'Part', 'null');
END_IF

IF __ISVALIDREF(PositionInfo) THEN
	TempString := LREAL_TO_FMTSTR(PositionInfo.fTrackPosition, 3, TRUE);
	JsonParser.AddStringMember(XTSJsonObject, 'ActPos', TempString);
ELSE
	TempString := LREAL_TO_FMTSTR(_Axis.NcToPlc.ModuloActPos, 3, TRUE);
	JsonParser.AddStringMember(XTSJsonObject, 'ActPos', TempString);
END_IF

TempString := LREAL_TO_FMTSTR(_Axis.NcToPlc.ActVelo, 3, TRUE);
JsonParser.AddStringMember(XTSJsonObject, 'ActVel', TempString);
TempString := LREAL_TO_FMTSTR(_Axis.NcToPlc.PosDiff, 3, TRUE);
JsonParser.AddStringMember(XTSJsonObject, 'PosLag', TempString);
JsonParser.AddObjectMember(XTSJsonObject, 'MoveDetails');
XTSJsonObject := JsonParser.FindMember(XTSJsonObject, 'MoveDetails');
TempString	  := LREAL_TO_FMTSTR(Position, 3, TRUE);
JsonParser.AddStringMember(XTSJsonObject, 'P', TempString);
IF Velocity = MC_DEFAULT THEN
	TempString := LREAL_TO_FMTSTR(0.0, 1, TRUE);
ELSE
	TempString := LREAL_TO_FMTSTR(Velocity, 3, TRUE);
END_IF

JsonParser.AddStringMember(XTSJsonObject, 'V', TempString);

// TempString := LREAL_TO_FMTSTR(Acceleration, 3, TRUE);
IF Acceleration = MC_DEFAULT THEN
	TempString := LREAL_TO_FMTSTR(0.0, 1, TRUE);
ELSE
	TempString := LREAL_TO_FMTSTR(Acceleration, 3, TRUE);
END_IF

JsonParser.AddStringMember(XTSJsonObject, 'A', TempString);
IF Acceleration = MC_DEFAULT THEN
	TempString := LREAL_TO_FMTSTR(0.0, 1, TRUE);
ELSE
	TempString := LREAL_TO_FMTSTR(Deceleration, 3, TRUE);
END_IF

// TempString := LREAL_TO_FMTSTR(Deceleration, 3, TRUE);
JsonParser.AddStringMember(XTSJsonObject, 'D', TempString);
IF Gap = MC_DEFAULT THEN
	TempString := LREAL_TO_FMTSTR(0.0, 1, TRUE);
ELSE
	TempString := LREAL_TO_FMTSTR(Gap, 3, TRUE);
END_IF

// TempString := LREAL_TO_FMTSTR(Gap, 3, TRUE);
JsonParser.AddStringMember(XTSJsonObject, 'G', TempString);
Message := CONCAT(MoveType, ' commanded');
TraceWithJson(Message, JsonParser.GetJson(Document));
END_METHOD

METHOD PRIVATE TraceWriteBoolParameter
VAR_INPUT
	ParameterNumber : MC_AxisParameter;
	Value			: BOOL;
END_VAR

VAR
	Message		  : T_MaxString;
	Document	  : SJsonValue;
	XTSJsonObject : SJsonValue;
	TempString	  : T_MaxString;
	JsonAttribute : T_MaxString;
END_VAR
{analysis -62}
Document := JsonParser.NewDocument();
JsonParser.AddObjectMember(Document, 'Mover');
XTSJsonObject := JsonParser.FindMember(Document, 'Mover');
JsonParser.AddUintMember(XTSJsonObject, 'AxisID', Axis.NcToPlc.AxisId);
IF ipMover <> 0 THEN
	TempString := ipMover.GetObjectName();
	JsonParser.AddStringMember(XTSJsonObject, 'Name', TempString);
END_IF

IF ipCurrentTrack <> 0 THEN
	TempString := ipCurrentTrack.Name;
	JsonParser.AddStringMember(XTSJsonObject, 'Track', TempString);
ELSE
	JsonParser.AddStringMember(XTSJsonObject, 'Track', 'null');
END_IF

IF ipCurrentPart <> 0 THEN
	TempString := ipCurrentPart.Name;
	JsonParser.AddStringMember(XTSJsonObject, 'Part', TempString);
ELSE
	JsonParser.AddStringMember(XTSJsonObject, 'Part', 'null');
END_IF

IF __ISVALIDREF(PositionInfo) THEN
	TempString := LREAL_TO_FMTSTR(PositionInfo.fTrackPosition, 3, TRUE);
	JsonParser.AddStringMember(XTSJsonObject, 'ActPos', TempString);
ELSE
	TempString := LREAL_TO_FMTSTR(_Axis.NcToPlc.ModuloActPos, 3, TRUE);
	JsonParser.AddStringMember(XTSJsonObject, 'ActPos', TempString);
END_IF

TempString := LREAL_TO_FMTSTR(_Axis.NcToPlc.ActVelo, 3, TRUE);
JsonParser.AddStringMember(XTSJsonObject, 'ActVel', TempString);
TempString := LREAL_TO_FMTSTR(_Axis.NcToPlc.PosDiff, 3, TRUE);
JsonParser.AddStringMember(XTSJsonObject, 'PosLag', TempString);
JsonParser.AddObjectMember(XTSJsonObject, 'Param');
XTSJsonObject := JsonParser.FindMember(XTSJsonObject, 'Param');
JsonParser.AddUintMember(XTSJsonObject, 'Parameter', TO_UINT(ParameterNumber));
JsonParser.AddBoolMember(XTSJsonObject, 'Value', Value);
Message := 'WriteBoolParameter commanded';
TraceWithJson(Message, JsonParser.GetJson(Document));
END_METHOD

METHOD PRIVATE TraceWriteParameter
VAR_INPUT
	ParameterNumber : MC_AxisParameter;
	Value			: LREAL;
END_VAR

VAR
	Message		  : T_MaxString;
	Document	  : SJsonValue;
	XTSJsonObject : SJsonValue;
	TempString	  : T_MaxString;
	JsonAttribute : T_MaxString;
END_VAR
{analysis -62}
Document := JsonParser.NewDocument();
JsonParser.AddObjectMember(Document, 'Mover');
XTSJsonObject := JsonParser.FindMember(Document, 'Mover');
JsonParser.AddUintMember(XTSJsonObject, 'AxisID', Axis.NcToPlc.AxisId);
IF ipMover <> 0 THEN
	TempString := ipMover.GetObjectName();
	JsonParser.AddStringMember(XTSJsonObject, 'Name', TempString);
END_IF

IF ipCurrentTrack <> 0 THEN
	TempString := ipCurrentTrack.Name;
	JsonParser.AddStringMember(XTSJsonObject, 'Track', TempString);
ELSE
	JsonParser.AddStringMember(XTSJsonObject, 'Track', 'null');
END_IF

IF ipCurrentPart <> 0 THEN
	TempString := ipCurrentPart.Name;
	JsonParser.AddStringMember(XTSJsonObject, 'Part', TempString);
ELSE
	JsonParser.AddStringMember(XTSJsonObject, 'Part', 'null');
END_IF

IF __ISVALIDREF(PositionInfo) THEN
	TempString := LREAL_TO_FMTSTR(PositionInfo.fTrackPosition, 3, TRUE);
	JsonParser.AddStringMember(XTSJsonObject, 'ActPos', TempString);
ELSE
	TempString := LREAL_TO_FMTSTR(_Axis.NcToPlc.ModuloActPos, 3, TRUE);
	JsonParser.AddStringMember(XTSJsonObject, 'ActPos', TempString);
END_IF

TempString := LREAL_TO_FMTSTR(_Axis.NcToPlc.ActVelo, 3, TRUE);
JsonParser.AddStringMember(XTSJsonObject, 'ActVel', TempString);
TempString := LREAL_TO_FMTSTR(_Axis.NcToPlc.PosDiff, 3, TRUE);
JsonParser.AddStringMember(XTSJsonObject, 'PosLag', TempString);
JsonParser.AddObjectMember(XTSJsonObject, 'Param');
XTSJsonObject := JsonParser.FindMember(XTSJsonObject, 'Param');
JsonParser.AddUintMember(XTSJsonObject, 'Parameter', TO_UINT(ParameterNumber));
JsonParser.AddDoubleMember(XTSJsonObject, 'Value', Value);
Message := 'WriteParameter commanded';
TraceWithJson(Message, JsonParser.GetJson(Document));
END_METHOD

PROPERTY AxisRefLinked : BOOL
GET
IF F_GetMappingStatus(ADR(_Axis.NcToPlc), SIZEOF(_Axis.NcToPlc)) <> EPlcMappingStatus.MS_Mapped THEN
	AxisRefLinked := FALSE;
	RETURN;
END_IF

IF F_GetMappingStatus(ADR(_Axis.PlcToNc), SIZEOF(_Axis.PlcToNc)) <> EPlcMappingStatus.MS_Mapped THEN
	AxisRefLinked := FALSE;
	RETURN;
END_IF

AxisRefLinked := TRUE;
END_GET
END_PROPERTY

PROPERTY CurrentPart : I_XTS_Part
GET
CurrentPart := ipCurrentPart;
END_GET
SET
ipCurrentPart := CurrentPart;
END_SET
END_PROPERTY

PROPERTY CurrentPartOID : OTCID
GET
IF __ISVALIDREF(PositionInfo) THEN
	CurrentPartOID := PositionInfo.nPartObjectid;
END_IF
END_GET
END_PROPERTY

PROPERTY CurrentTrack : I_XTS_Track
GET
CurrentTrack := ipCurrentTrack;
END_GET
SET
ipCurrentTrack := CurrentTrack;
END_SET
END_PROPERTY

PROPERTY CurrentTrackOID : OTCID
GET
IF __ISVALIDREF(PositionInfo) THEN
	CurrentTrackOID := PositionInfo.nTrackObjectid;
END_IF
END_GET
END_PROPERTY

METHOD FB_reinit : BOOL
VAR_INPUT
END_VAR
MCMoveAbsoluteCA := RingBuffer_MCMoveAbsoluteCA.CurrentFB;
MCMoveRelativeCA := RingBuffer_MCMoveRelativeCA.CurrentFB;
END_METHOD

PROPERTY Group : REFERENCE TO AXES_GROUP_REF
GET
Group REF= _Group;
END_GET
SET
_Group REF= Group;
END_SET
END_PROPERTY

METHOD PROTECTED Initialize : BOOL
CASE InitializeState OF
	E_InitializeState_Mover.eInitializeStateMover_Check:
		IF ipMover <> 0 AND __ISVALIDREF(_Group) THEN
			InitializeState := E_InitializeState_Mover.eInitializeStateMover_GetSoftDriveInterfaces;
		ELSIF NOT (ipMover <> 0) THEN
			IF Parameters_XTS.ENABLE_DEBUG_TRACING THEN
				Trace('Mover initialization attempted with null reference');
			END_IF

			InitializeState := InitializeState := E_InitializeState_Mover.eInitializeStateMover_Failed;
		ELSIF NOT __ISVALIDREF(_Group) THEN
			IF Parameters_XTS.ENABLE_DEBUG_TRACING THEN
				Trace('Mover initialization attempted with no CA group set');
			END_IF

			InitializeState := InitializeState := E_InitializeState_Mover.eInitializeStateMover_Failed;
		END_IF

	E_InitializeState_Mover.eInitializeStateMover_GetSoftDriveInterfaces:
		ipSoftDrive := ipMover.SoftDrive;
		IF ipSoftDrive <> 0 THEN
			IF NOT ipSoftDrive.P_IsInitialized THEN
				IF Parameters_XTS.ENABLE_DEBUG_TRACING THEN
					Trace('SoftDrive is not initialized.');
				END_IF

				InitializeState := E_InitializeState_Mover.eInitializeStateMover_Failed;
				RETURN;
			END_IF
		ELSE
			IF Parameters_XTS.ENABLE_DEBUG_TRACING THEN
				Trace('SoftDrive did not return a valid interface');
			END_IF

			InitializeState := E_InitializeState_Mover.eInitializeStateMover_Failed;
			RETURN;
		END_IF

		InitializeState := E_InitializeState_Mover.eInitializeStateMover_GetSoftDriveInterfaces_Encoder;

	E_InitializeState_Mover.eInitializeStateMover_GetSoftDriveInterfaces_Encoder:
		ipEncoder := ipSoftDrive.Encoder;
		IF ipEncoder <> 0 THEN
			IF NOT ipEncoder.P_IsInitialized THEN
				IF Parameters_XTS.ENABLE_DEBUG_TRACING THEN
					Trace('SoftDrive Encoder is not initialized.');
				END_IF

				InitializeState := E_InitializeState_Mover.eInitializeStateMover_Failed;
				RETURN;
			END_IF
		ELSE
			IF Parameters_XTS.ENABLE_DEBUG_TRACING THEN
				Trace('SoftDrive Encoder did not return a valid interface');
			END_IF

			InitializeState := E_InitializeState_Mover.eInitializeStateMover_Failed;
			RETURN;
		END_IF

		InitializeState := E_InitializeState_Mover.eInitializeStateMover_GetSoftDriveInterfaces_FeedForward;

	E_InitializeState_Mover.eInitializeStateMover_GetSoftDriveInterfaces_FeedForward:
		ipFeedForward := ipSoftDrive.FeedForward;
		IF ipFeedForward <> 0 THEN
			IF NOT ipFeedForward.P_IsInitialized THEN
				IF Parameters_XTS.ENABLE_DEBUG_TRACING THEN
					Trace('SoftDrive FeedForward number is not initialized.');
				END_IF

				InitializeState := E_InitializeState_Mover.eInitializeStateMover_Failed;
				RETURN;
			END_IF
		ELSE
			IF Parameters_XTS.ENABLE_DEBUG_TRACING THEN
				Trace('SoftDrive FeedForward did not return a valid interface');
			END_IF

			InitializeState := E_InitializeState_Mover.eInitializeStateMover_Failed;
			RETURN;
		END_IF

		InitializeState := E_InitializeState_Mover.eInitializeStateMover_GetSoftDriveInterfaces_Filters;

	E_InitializeState_Mover.eInitializeStateMover_GetSoftDriveInterfaces_Filters:
		ipFilter1 := ipSoftDrive.Filter1;
		IF ipFilter1 <> 0 THEN
			IF NOT ipFilter1.P_IsInitialized THEN
				IF Parameters_XTS.ENABLE_DEBUG_TRACING THEN
					Trace('SoftDrive Filter 1 is not initialized.');
				END_IF

				InitializeState := E_InitializeState_Mover.eInitializeStateMover_Failed;
				RETURN;
			END_IF
		ELSE
			IF Parameters_XTS.ENABLE_DEBUG_TRACING THEN
				Trace('SoftDrive Filter 1 did not return a valid interface');
			END_IF

			InitializeState := E_InitializeState_Mover.eInitializeStateMover_Failed;
			RETURN;
		END_IF

		ipFilter2 := ipSoftDrive.Filter2;
		IF ipFilter2 <> 0 THEN
			IF NOT ipFilter2.P_IsInitialized THEN
				IF Parameters_XTS.ENABLE_DEBUG_TRACING THEN
					Trace('SoftDrive Filter 2 is not initialized.');
				END_IF
			END_IF
		ELSE
			IF Parameters_XTS.ENABLE_DEBUG_TRACING THEN
				Trace('SoftDrive Filter 2 did not return a valid interface');
			END_IF
		END_IF

		InitializeState := E_InitializeState_Mover.eInitializeStateMover_GetSoftDriveInterfaces_Interpolator;

	E_InitializeState_Mover.eInitializeStateMover_GetSoftDriveInterfaces_Interpolator:
		ipInterpolator := ipSoftDrive.Interpolator;
		IF ipInterpolator <> 0 THEN
			IF NOT ipInterpolator.P_IsInitialized THEN
				IF Parameters_XTS.ENABLE_DEBUG_TRACING THEN
					Trace('SoftDrive Interpolator is not initialized.');
				END_IF

				InitializeState := E_InitializeState_Mover.eInitializeStateMover_Failed;
				RETURN;
			END_IF
		ELSE
			IF Parameters_XTS.ENABLE_DEBUG_TRACING THEN
				Trace('SoftDrive Interpolator did not return a valid interface');
			END_IF

			InitializeState := E_InitializeState_Mover.eInitializeStateMover_Failed;
			RETURN;
		END_IF

		InitializeState := E_InitializeState_Mover.eInitializeStateMover_GetSoftDriveInterfaces_PositionController;

	E_InitializeState_Mover.eInitializeStateMover_GetSoftDriveInterfaces_PositionController:
		ipPositionController := ipSoftDrive.PositionControl;
		IF ipPositionController <> 0 THEN
			IF NOT ipPositionController.P_IsInitialized THEN
				IF Parameters_XTS.ENABLE_DEBUG_TRACING THEN
					Trace('SoftDrive Position Controller is not initialized.');
				END_IF

				InitializeState := E_InitializeState_Mover.eInitializeStateMover_Failed;
				RETURN;
			END_IF
		ELSE
			IF Parameters_XTS.ENABLE_DEBUG_TRACING THEN
				Trace('SoftDrive Position Controller did not return a valid interface');
			END_IF

			InitializeState := E_InitializeState_Mover.eInitializeStateMover_Failed;
			RETURN;
		END_IF

		InitializeState := E_InitializeState_Mover.eInitializeStateMover_GetSoftDriveInterfaces_VelocityController;

	E_InitializeState_Mover.eInitializeStateMover_GetSoftDriveInterfaces_VelocityController:
		ipVelocityController := ipSoftDrive.VelocityControl;
		IF ipVelocityController <> 0 THEN
			IF NOT ipVelocityController.P_IsInitialized THEN
				IF Parameters_XTS.ENABLE_DEBUG_TRACING THEN
					Trace('SoftDrive Velocity Controller is not initialized.');
				END_IF

				InitializeState := E_InitializeState_Mover.eInitializeStateMover_Failed;
				RETURN;
			END_IF
		ELSE
			IF Parameters_XTS.ENABLE_DEBUG_TRACING THEN
				Trace('SoftDrive Velocity Controller did not return a valid interface');
			END_IF

			InitializeState := E_InitializeState_Mover.eInitializeStateMover_Failed;
			RETURN;
		END_IF

		InitializeState := E_InitializeState_Mover.eInitializeStateMover_ReadTcIOParameters;

	//TODO:	
	E_InitializeState_Mover.eInitializeStateMover_ReadTcIOParameters:
		PositionInfo	REF= ipMover.GetPositionInfo();
		InitializeState := E_InitializeState_Mover.eInitializeStateMover_CheckDriveLinks;

	E_InitializeState_Mover.eInitializeStateMover_CheckDriveLinks:
		// Verify that the AXIS_REF is actually linked with the NC
		IF F_GetMappingStatus(ADR(_Axis.NcToPlc), SIZEOF(_Axis.NcToPlc)) <> EPlcMappingStatus.MS_Mapped THEN
			IF NOT Parameters_XTS.ALLOW_UNLINKED_MOVER_NC_AXES THEN
				IF Parameters_XTS.ENABLE_DEBUG_TRACING THEN
					Trace('NC axis is not linked!');
				END_IF

				InitializeState := E_InitializeState_Mover.eInitializeStateMover_Failed;
				RETURN;
			END_IF
		END_IF

		IF F_GetMappingStatus(ADR(_Axis.PlcToNc), SIZEOF(_Axis.PlcToNc)) <> EPlcMappingStatus.MS_Mapped THEN
			IF NOT Parameters_XTS.ALLOW_UNLINKED_MOVER_NC_AXES THEN
				IF Parameters_XTS.ENABLE_DEBUG_TRACING THEN
					Trace('NC axis is not linked!');
				END_IF

				InitializeState := E_InitializeState_Mover.eInitializeStateMover_Failed;
				RETURN;
			END_IF
		END_IF

		// AxisId will be populated by the NC when it finishes starting

		// This prevents requesting motion before NC Init/nuisance errors
		IF _Axis.NcToPlc.AxisId = 0 THEN
			IF NOT Parameters_XTS.ALLOW_UNLINKED_MOVER_NC_AXES THEN
				IF Parameters_XTS.ENABLE_DEBUG_TRACING THEN
					Trace('NC axis ID has not been set. Check axis links?');
				END_IF

				InitializeState := E_InitializeState_Mover.eInitializeStateMover_Failed;
				RETURN;
			END_IF
		END_IF

		InitializeState := E_InitializeState_Mover.eInitializeStateMover_ReadNCParameters;

	E_InitializeState_Mover.eInitializeStateMover_ReadNCParameters:
		// Read all NC parameters
		IF Parameters_XTS.ALLOW_UNLINKED_MOVER_NC_AXES THEN
			InitializeState := E_InitializeState_Mover.eInitializeStateMover_Complete;
		ELSE
			MCReadParameterSet(Parameter := _AxisParameters, Axis := _Axis, Execute := TRUE);
			IF NOT MCReadParameterSet.Busy THEN
				IF MCReadParameterSet.Error THEN
					_Error			:= TRUE;
					_ErrorID		:= MCReadParameterSet.ErrorID;
					InitializeState := E_InitializeState_Mover.eInitializeStateMover_Failed;
				ELSIF MCReadParameterSet.Done THEN
					_Velocity		:= _AxisParameters.fVeloSlowManual;
					_Acceleration	:= _AxisParameters.fAcceleration;
					_Deceleration	:= _AxisParameters.fDeceleration;
					_Jerk			:= _AxisParameters.fJerk;
					SoftDriveMode.8 := TRUE; // Set default SoftDrive mode to Position Mode
					InitializeState := E_InitializeState_Mover.eInitializeStateMover_Complete;
				END_IF

				MCReadParameterSet(Parameter := _AxisParameters, Axis := _Axis, Execute := FALSE);
			END_IF
		END_IF

	E_InitializeState_Mover.eInitializeStateMover_Complete:
		_Busy	   := FALSE;
		Initialize := TRUE;

	E_InitializeState_Mover.eInitializeStateMover_Failed:
		_Busy  := FALSE;
		_Error := TRUE;
END_CASE
END_METHOD

END_FUNCTION_BLOCK

// Parts/I_XTS_Part
INTERFACE I_XTS_Part

PROPERTY Name : STRING
GET
END_GET
END_PROPERTY

PROPERTY ReadyToEnable : BOOL
GET
END_GET
END_PROPERTY

END_INTERFACE

// Tracks/I_XTS_Track
INTERFACE I_XTS_Track

METHOD GetTrackPositionByPart
VAR_INPUT
	Position : LREAL;
	Part	 : OTCID;
END_VAR

VAR_OUTPUT
	TrackPosition : LREAL;
END_VAR
END_METHOD

PROPERTY IsClosed : BOOL
GET
END_GET
END_PROPERTY

PROPERTY Length : LREAL
GET
END_GET
END_PROPERTY

PROPERTY Name : STRING
GET
END_GET
END_PROPERTY

END_INTERFACE

// Utilities/FB_RingBuffer_MCMoveRelativeCA
FUNCTION_BLOCK FB_RingBuffer_MCMoveRelativeCA
VAR CONSTANT
	MAX_FB_COUNT : UDINT := 1;
END_VAR

VAR_IN_OUT
	Axis : AXIS_REF;
END_VAR

VAR_OUTPUT
END_VAR

VAR
	MCMoveRelativeCA : ARRAY[0..MAX_FB_COUNT] OF MC_MoveRelativeCA;
	FBIndex			 : UDINT;
	i				 : UDINT;
END_VAR

(* This buffer ensures you always have a clean FB to use for a move *)

FOR i := 0 TO MAX_FB_COUNT DO
	MCMoveRelativeCA[i](Axis := Axis);
END_FOR

PROPERTY CurrentFB : POINTER TO MC_MoveAbsoluteCA
GET
CurrentFB := ADR(MCMoveRelativeCA[FBIndex]);
END_GET
END_PROPERTY

METHOD GetNewFB : POINTER TO MC_MoveAbsoluteCA
VAR_INPUT
END_VAR
FBIndex := FBIndex + 1;
IF FBIndex > MAX_FB_COUNT THEN
	MCMoveRelativeCA[MAX_FB_COUNT].Execute := FALSE;
	FBIndex								   := 0;
ELSE
	MCMoveRelativeCA[FBIndex - 1].Execute := FALSE;
END_IF

GetNewFB := ADR(MCMoveRelativeCA[FBIndex]);
END_METHOD

END_FUNCTION_BLOCK

// Utilities/FB_RingBuffer_MCMoveAbsoluteCA
FUNCTION_BLOCK FB_RingBuffer_MCMoveAbsoluteCA
VAR CONSTANT
	MAX_FB_COUNT : UDINT := 1;
END_VAR

VAR_IN_OUT
	Axis : AXIS_REF;
END_VAR

VAR_OUTPUT
END_VAR

VAR
	MCMoveAbsoluteCA : ARRAY[0..MAX_FB_COUNT] OF MC_MoveAbsoluteCA;
	FBIndex			 : UDINT;
	i				 : UDINT;
END_VAR

(* This buffer ensures you always have a clean FB to use for a move *)

FOR i := 0 TO MAX_FB_COUNT DO
	MCMoveAbsoluteCA[i](Axis := Axis);
END_FOR

PROPERTY CurrentFB : POINTER TO MC_MoveAbsoluteCA
GET
CurrentFB := ADR(MCMoveAbsoluteCA[FBIndex]);
END_GET
END_PROPERTY

METHOD GetNewFB : POINTER TO MC_MoveAbsoluteCA
VAR_INPUT
END_VAR
FBIndex := FBIndex + 1;
IF FBIndex > MAX_FB_COUNT THEN
	MCMoveAbsoluteCA[MAX_FB_COUNT].Execute := FALSE;
	FBIndex								   := 0;
ELSE
	MCMoveAbsoluteCA[FBIndex - 1].Execute := FALSE;
END_IF

GetNewFB := ADR(MCMoveAbsoluteCA[FBIndex]);
END_METHOD

END_FUNCTION_BLOCK

// Utilities/FB_RingBuffer_MCGearInPosCA
FUNCTION_BLOCK FB_RingBuffer_MCGearInPosCA
VAR CONSTANT
	MAX_FB_COUNT : UDINT := 1;
END_VAR

VAR_IN_OUT
	Master : AXIS_REF;
	Slave  : AXIS_REF;
END_VAR

VAR_OUTPUT
END_VAR

VAR
	MGearInPosCA : ARRAY[0..MAX_FB_COUNT] OF MC_GearInPosCA;
	FBIndex		 : UDINT;
	i			 : UDINT;
END_VAR

(* This buffer ensures you always have a clean FB to use for a move *)

FOR i := 0 TO MAX_FB_COUNT DO
	MGearInPosCA[i](Master := Master, Slave := Slave);
END_FOR

PROPERTY CurrentFB : POINTER TO MC_GearInPosCA
GET
CurrentFB := ADR(MGearInPosCA[FBIndex]);
END_GET
END_PROPERTY

METHOD GetNewFB : POINTER TO MC_GearInPosCA
VAR_INPUT
END_VAR
FBIndex := FBIndex + 1;
IF FBIndex > MAX_FB_COUNT THEN
	MGearInPosCA[MAX_FB_COUNT].Execute := FALSE;
	FBIndex							   := 0;
ELSE
	MGearInPosCA[FBIndex - 1].Execute := FALSE;
END_IF

GetNewFB := ADR(MGearInPosCA[FBIndex]);
END_METHOD

END_FUNCTION_BLOCK

// Parts/FB_XTS_Part
FUNCTION_BLOCK INTERNAL FINAL FB_XTS_Part EXTENDS FB_CyclicFB IMPLEMENTS I_XTS_Part
VAR_INPUT
	OID	   : OTCID;
	ipXPU  : I_XTS_Xpu;
	ipPart : I_TcIoXtsXpuPart;
END_VAR

VAR
	NumberOfModules		 : UDINT;
	NumberOfControlAreas : UDINT;
	ipModules_CoE		 : ARRAY[1..TcIoXtsEnvironmentParameterList.MaxModulesPerPart] OF I_AT2xxxXtsMotor;
	ipModules_TcIo		 : ARRAY[1..TcIoXtsEnvironmentParameterList.MaxModulesPerPart] OF I_TcIoXtsPartModule;
	ipControlAreas		 : ARRAY[1..TcIoXtsEnvironmentParameterList.MaxAreasPerPart] OF I_TcIoXtsPartControlArea;
	InitializeState		 : E_InitializeState_Part;
	ModuleCoEIndex		 : UDINT := 1;
	PartDriveState		 : DriveState;
	_ModuleCoEData		 : ARRAY[1..TcIoXtsEnvironmentParameterList.MaxModulesPerPart] OF ST_AT2xxxAllCoEData;
	_ReadyToEnable		 : BOOL;
END_VAR

METHOD PUBLIC CyclicLogic
VAR
	CurrentModuleCoEData : REFERENCE TO ST_AT2xxxAllCoEData;
	i					 : UDINT;
END_VAR
IF NOT _InitComplete THEN
	_InitComplete := Initialize();
	RETURN;
END_IF

IF ipXPU.InSimulationMode THEN
	_ReadyToEnable := TRUE;
	PartDriveState := DriveState.Unknown;
ELSE
	PartDriveState := ipPart.GetDriveState();
	CASE PartDriveState OF
		DriveState.Unknown:
			_ReadyToEnable := FALSE;

		DriveState.FaultReactionActive:
			_ReadyToEnable := FALSE;

		DriveState.Fault:
			_ReadyToEnable := FALSE;

		DriveState.NotReadyToSwitchOn:
			_ReadyToEnable := FALSE;

		DriveState.SwitchOnDisabled:
			_ReadyToEnable := FALSE;

		DriveState.ReadyToSwitchOn:
			_ReadyToEnable := TRUE;

		DriveState.SwitchedOn:
			_ReadyToEnable := TRUE;

		DriveState.OperationEnabled:
			_ReadyToEnable := TRUE;

	ELSE
		_ReadyToEnable := FALSE;
	END_CASE

	FOR i := 1 TO NumberOfModules DO
		IF ipModules_CoE[i].AllCoE.UpdateAllCoEData() THEN
			CurrentModuleCoEData REF= ipModules_CoE[i].AllCoE.AllCoEData;
			MEMCPY(ADR(_ModuleCoEData[i]), ADR(CurrentModuleCoEData), SIZEOF(ST_AT2xxxAllCoEData));
		END_IF
	END_FOR
END_IF

_Error := PartDriveState = DriveState.Fault;
END_METHOD

METHOD PRIVATE Initialize : BOOL
VAR
	i : UDINT;
END_VAR
CASE InitializeState OF
	E_InitializeState_Part.eInitializeStatePart_Check:
		IF ipPart <> 0 AND ipXPU <> 0 THEN
			InitializeState := E_InitializeState_Part.eInitializeStatePart_GetModuleInterfaces;
		ELSE
			IF Parameters_XTS.ENABLE_DEBUG_TRACING THEN
				Trace('Part initialization attempted with null reference');
			END_IF

			InitializeState := E_InitializeState_Part.eInitializeStatePart_Failed;
		END_IF

	E_InitializeState_Part.eInitializeStatePart_GetModuleInterfaces:
		NumberOfModules := ipPart.GetModuleCount();
		IF NumberOfModules > 0 THEN
			FOR i := 1 TO NumberOfModules DO
				ipModules_CoE[i]  := ipPart.ModuleCoE(TO_UINT(i));
				ipModules_TcIo[i] := ipPart.ModuleTcIo(TO_UINT(i));
				IF ipModules_CoE[i] <> 0 THEN
					;
				ELSE
					IF Parameters_XTS.ENABLE_DEBUG_TRACING THEN
						Trace(CONCAT('Module number (CoE) ', CONCAT(TO_STRING(i), ' did not return a valid interface')));
					END_IF

					InitializeState := E_InitializeState_Part.eInitializeStatePart_Failed;
					RETURN;
				END_IF

				IF ipModules_TcIo[i] <> 0 THEN
					IF NOT ipModules_TcIo[i].P_IsInitialized THEN
						IF Parameters_XTS.ENABLE_DEBUG_TRACING THEN
							Trace(CONCAT('Module number (TcIo) ', CONCAT(TO_STRING(i), ' is not initialized.')));
						END_IF

						InitializeState := E_InitializeState_Part.eInitializeStatePart_Failed;
						RETURN;
					END_IF
				ELSE
					IF Parameters_XTS.ENABLE_DEBUG_TRACING THEN
						Trace(CONCAT('Module number (TcIo) ', CONCAT(TO_STRING(i), ' did not return a valid interface')));
					END_IF

					InitializeState := E_InitializeState_Part.eInitializeStatePart_Failed;
					RETURN;
				END_IF
			END_FOR
		END_IF

		InitializeState := E_InitializeState_Part.eInitializeStatePart_GetControlAreaInterfaces;

	E_InitializeState_Part.eInitializeStatePart_GetControlAreaInterfaces:
		NumberOfControlAreas := ipPart.GetAreaCount();
		IF NumberOfControlAreas > 0 THEN
			FOR i := 1 TO NumberOfControlAreas DO
				ipControlAreas[i] := ipPart.ControlAreaTcIo(TO_UINT(i));
				IF ipControlAreas[i] <> 0 THEN
					IF NOT ipControlAreas[i].P_IsInitialized THEN
						IF Parameters_XTS.ENABLE_DEBUG_TRACING THEN
							Trace(CONCAT('Control area ', CONCAT(TO_STRING(i), ' is not initialized.')));
						END_IF

						InitializeState := E_InitializeState_Part.eInitializeStatePart_Failed;
						RETURN;
					END_IF
				ELSE
					IF Parameters_XTS.ENABLE_DEBUG_TRACING THEN
						Trace(CONCAT('Control area ', CONCAT(TO_STRING(i), ' did not return a valid interface')));
					END_IF

					InitializeState := E_InitializeState_Part.eInitializeStatePart_Failed;
					RETURN;
				END_IF
			END_FOR
		END_IF

		InitializeState := E_InitializeState_Part.eInitializeStatePart_Complete;

	E_InitializeState_Part.eInitializeStatePart_Complete:
		_Busy	   := FALSE;
		Initialize := TRUE;

	E_InitializeState_Part.eInitializeStatePart_Failed:
		_Busy  := FALSE;
		_Error := TRUE;
END_CASE
END_METHOD

PROPERTY ModuleCoEData : ARRAY[1..TcIoXtsEnvironmentParameterList.MaxModulesPerPart] OF ST_AT2xxxAllCoEData
GET
ModuleCoEData := _ModuleCoEData;
END_GET
END_PROPERTY

PROPERTY Name : STRING
GET
IF ipPart <> 0 THEN
	Name := ipPart.GetObjectName();
END_IF
END_GET
END_PROPERTY

PROPERTY ReadyToEnable : BOOL
GET
ReadyToEnable := _ReadyToEnable;
END_GET
END_PROPERTY

METHOD PUBLIC Reset : BOOL
IF (ipPart <> 0) THEN
	Reset := ipPart.TriggerReset();
END_IF
END_METHOD

END_FUNCTION_BLOCK

// XPU/I_XTS_Xpu
INTERFACE I_XTS_Xpu

METHOD GetPositionOnTrack : LREAL
VAR_INPUT
	TrackID	 : OTCID;
	PartID	 : OTCID;
	Position : LREAL;
END_VAR
END_METHOD

METHOD GiveMover : BOOL
VAR_INPUT
	RequestingStation : I_XTS_StationNeighbor;
END_VAR
END_METHOD

PROPERTY InSimulationMode : BOOL
GET
END_GET
END_PROPERTY

END_INTERFACE

// Stations/I_XTS_StationNeighbor
INTERFACE I_XTS_StationNeighbor

METHOD GiveMover : BOOL
VAR_INPUT
	RequestingStation : I_XTS_StationNeighbor;
END_VAR
END_METHOD

PROPERTY StationName : STRING
GET
END_GET
END_PROPERTY

METHOD TakeMover : BOOL
VAR_INPUT
	Mover : I_XTS_Mover;
END_VAR
END_METHOD

END_INTERFACE

// Project Information/F_GetCompany
// This function has been automatically generated from the project information.
{attribute 'signature_flag' := '1073741824'}
{attribute 'TcGenerated'}
{attribute 'no-analysis'}
FUNCTION F_GetCompany : WSTRING
VAR_INPUT
END_VAR

F_GetCompany := "Beckhoff Automation LLC";

END_FUNCTION

// Project Information/F_GetTitle
// This function has been automatically generated from the project information.
{attribute 'signature_flag' := '1073741824'}
{attribute 'TcGenerated'}
{attribute 'no-analysis'}
FUNCTION F_GetTitle : WSTRING
VAR_INPUT
END_VAR

F_GetTitle := "SPT XTS";

END_FUNCTION

// Project Information/F_GetVersion
// This function has been automatically generated from the project information.
{attribute 'signature_flag' := '1073741824'}
{attribute 'TcGenerated'}
{attribute 'no-analysis'}
FUNCTION F_GetVersion : ST_LibVersion
VAR_INPUT
END_VAR

F_GetVersion.iMajor	   := 4;
F_GetVersion.iMinor	   := 0;
F_GetVersion.iBuild	   := 0;
F_GetVersion.iRevision := 0;
F_GetVersion.sVersion  := '4.0.0';
F_GetVersion.nFlags	   := 1;

END_FUNCTION

// Stations/FB_XTS_InfoStation
FUNCTION_BLOCK INTERNAL FINAL FB_XTS_InfoStation EXTENDS FB_CyclicFB IMPLEMENTS I_XTS_InfoStation, I_XTS_StationNeighbor
VAR_INPUT
	ipInfoStation : I_TcIoXtsInfoServerInfoStation;
	ipXPU		  : I_XTS_Xpu;
END_VAR

VAR
	InitializeState : E_InitializeState_Station;
	_MoverQueue		: FB_MoverQueue;
	ipStation		: I_XTS_ApplicationStation;
	MoversAssigned	: ARRAY[1..TcIoXtsEnvironmentParameterList.MaxXtsMoversPerXpu] OF UDINT;
END_VAR

METHOD PUBLIC CyclicLogic
VAR
END_VAR
IF NOT _InitComplete THEN
	_InitComplete := Initialize();
	RETURN;
END_IF
END_METHOD

PROPERTY ApplicationStation : I_XTS_ApplicationStation
GET
ApplicationStation := ipStation;
END_GET
SET
ipStation := ApplicationStation;
END_SET
END_PROPERTY

PROPERTY Color : E_Colors_ARGB
GET
IF ipInfoStation <> 0 THEN
	Color := ipInfoStation.GetStationColor();
END_IF
END_GET
SET
IF ipInfoStation <> 0 THEN
	ipInfoStation.SetStationColor(Color);
END_IF
END_SET
END_PROPERTY

METHOD PUBLIC GetMover : BOOL
IF ipXPU <> 0 THEN
	GetMover := ipXPU.GiveMover(THIS^);
END_IF
END_METHOD

METHOD PUBLIC GetStopPositionOnTrack : LREAL
VAR_INPUT
	TrackID	 : OTCID;
	Position : LREAL;
END_VAR

VAR
	PartOID				: OTCID;
	StartPositionOnPart : LREAL;
END_VAR
IF ipXPU <> 0 THEN
	PartOID				   := ipInfoStation.P_PartObjectIds[1];
	StartPositionOnPart	   := ipInfoStation.GetStartPositionOnPart();
	GetStopPositionOnTrack := ipXPU.GetPositionOnTrack(TrackID, PartOID, StartPositionOnPart + Position);
END_IF
END_METHOD

PROPERTY MoverQueue : REFERENCE TO FB_MoverQueue
GET
MoverQueue REF= _MoverQueue;
END_GET
END_PROPERTY

PROPERTY NumberOfStops : UDINT
GET
IF ipInfoStation <> 0 THEN
	NumberOfStops := ipInfoStation.GetStopPositionsCount();
END_IF
END_GET
END_PROPERTY

PROPERTY StopPositions : REFERENCE TO ARRAY[1..TcIoXtsEnvironmentParameterList.MaxXtsStopPositionsPerStation] OF LREAL
GET
IF ipInfoStation <> 0 THEN
	StopPositions REF= ipInfoStation.P_StopPositions;
END_IF
END_GET
END_PROPERTY

METHOD PUBLIC GiveMover : BOOL
VAR_INPUT
	RequestingStation : I_XTS_StationNeighbor;
END_VAR
// Station can release a mover
IF ipStation <> 0 THEN
	IF ipStation.CanReleaseMover THEN
		IF RequestingStation.TakeMover(_MoverQueue.FirstMover) THEN
			IF Parameters_XTS.ENABLE_DEBUG_TRACING THEN
				Trace(CONCAT('Passed Mover ', CONCAT(TO_STRING(_MoverQueue.FirstMover.MoverID), CONCAT(' from ', CONCAT(StationName, CONCAT(' to ', RequestingStation.StationName))))));
			END_IF

			_MoverQueue.Dequeue();
			GiveMover := TRUE;
		END_IF
	END_IF
END_IF
END_METHOD

PROPERTY StationName : STRING
GET
IF ipStation <> 0 THEN
	StationName := ipStation.Name;
ELSE
	StationName := '***UNKNOWN STATION***';
END_IF
END_GET
END_PROPERTY

METHOD PUBLIC TakeMover : BOOL
VAR_INPUT
	Mover : I_XTS_Mover;
END_VAR
// Check for valid interface pointer
IF ipStation <> 0 THEN
	IF ipStation.CanAcceptMover THEN
		IF Parameters_XTS.ENABLE_DEBUG_TRACING THEN
			Trace(CONCAT(StationName, CONCAT(' accepted Mover ', TO_STRING(Mover.MoverID))));
		END_IF

		Mover.Station := ipStation;
		TakeMover	  := _MoverQueue.Enqueue(Mover);
	END_IF
END_IF
END_METHOD

METHOD PRIVATE Initialize : BOOL
CASE InitializeState OF
	E_InitializeState_Station.eInitializeStateStation_Check:
		IF ipInfoStation <> 0 THEN
			InitializeState := E_InitializeState_Station.eInitializeStateStation_GetPartInfo;
		ELSE
			IF Parameters_XTS.ENABLE_DEBUG_TRACING THEN
				Trace('Station initialization attempted with null reference');
			END_IF

			InitializeState := E_InitializeState_Station.eInitializeStateStation_Failed;
		END_IF

	E_InitializeState_Station.eInitializeStateStation_GetPartInfo:
		IF ipInfoStation.GetPartCount() = 1 THEN
			InitializeState := E_InitializeState_Station.eInitializeStateStation_GetStopPositions;
		ELSE
			// Multiple parts per station not supported (yet)
			IF Parameters_XTS.ENABLE_DEBUG_TRACING THEN
				Trace('Multiple parts per station not supported...yet');
			END_IF

			InitializeState := E_InitializeState_Station.eInitializeStateStation_Failed;
		END_IF

	E_InitializeState_Station.eInitializeStateStation_GetStopPositions:
		IF ipInfoStation.GetStopPositionsCount() > 0 THEN
			InitializeState := E_InitializeState_Station.eInitializeStateStation_Complete;
		ELSE
			IF Parameters_XTS.ENABLE_DEBUG_TRACING THEN
				Trace('Station has no stop position');
			END_IF

			InitializeState := E_InitializeState_Station.eInitializeStateStation_Complete;
		END_IF

	E_InitializeState_Station.eInitializeStateStation_Complete:
		_Busy	   := FALSE;
		Initialize := TRUE;

	E_InitializeState_Station.eInitializeStateStation_Failed:
		_Busy  := FALSE;
		_Error := TRUE;
END_CASE
END_METHOD

PROPERTY IsAQueue : BOOL
GET
VAR
	StationConfig : ST_XTSStationConfig;
END_VAR
IF ipStation <> 0 THEN
	StationConfig := ipStation.Config;
	IsAQueue	  := StationConfig.IsAQueueStation;
END_IF
END_GET
END_PROPERTY

PROPERTY MoverIDsAssigned : ARRAY[1..TcIoXtsEnvironmentParameterList.MaxXtsMoversPerXpu] OF UDINT
GET
MoverIDsAssigned := _MoverQueue.MoverIDs;
END_GET
END_PROPERTY

// This method is called by HomeQueueStation via I_Mover. Clears mover FIFO and resets station sequences.
METHOD PUBLIC ReleaseAllMovers : BOOL
IF _MoverQueue.Count = 0 THEN
	ReleaseAllMovers := TRUE;
	RETURN;
ELSE
	ReleaseAllMovers := _MoverQueue.Clear();
END_IF
END_METHOD

PROPERTY StationID : UDINT
GET
IF ipInfoStation <> 0 THEN
	StationID := ipInfoStation.GetStationId();
END_IF
END_GET
END_PROPERTY

END_FUNCTION_BLOCK

// Tracks/FB_XTS_Track
FUNCTION_BLOCK INTERNAL FINAL FB_XTS_Track EXTENDS FB_CyclicFB IMPLEMENTS I_XTS_Track;
VAR_INPUT
	OID		: OTCID;
	ipTrack : I_TcIoXtsXpuTrack;
END_VAR

VAR
	NumberOfParts	: UDINT;
	Parts			: REFERENCE TO ARRAY[1..TcIoXtsEnvironmentParameterList.MaxPartsPerTrack] OF ST_PartInfoItems;
	InitializeState : E_InitializeState_Track;
END_VAR

METHOD PUBLIC CyclicLogic
VAR_INPUT
END_VAR
IF NOT _InitComplete THEN
	_InitComplete := Initialize();
	RETURN;
END_IF
END_METHOD

METHOD PUBLIC GetTrackPositionByPart
VAR_INPUT
	Position : LREAL;
	Part	 : OTCID;
END_VAR

VAR_OUTPUT
	TrackPosition : LREAL;
END_VAR

VAR
	i					   : UDINT;
	PartExists			   : BOOL;
	NumberOfPrecedingParts : UDINT;
	PrecedingPartDistance  : LREAL;
END_VAR
IF NOT (ipTrack <> 0) OR NOT __ISVALIDREF(Parts) THEN
	// Initialization not complete
	Trace('GetTrackPositionByPart() called before initialization!');
	_Error := TRUE;
	RETURN;
ELSIF Position < 0 OR Position > ipTrack.GetLength() THEN
	// Position outside of track
	Trace(CONCAT(TO_STRING(Position), CONCAT(' is outside of the track dimensions. Track: ', CONCAT(Name, CONCAT(' Length: ', TO_STRING(ipTrack.GetLength()))))));
	_Error := TRUE;
	RETURN;
ELSE
	_Error := FALSE;
END_IF

// Check if part is part of this track
FOR i := 1 TO ipTrack.GetPartCount() DO
	IF Parts[i].nObjectId = Part THEN
		TrackPosition := Parts[i].fOffset + Position;
		RETURN;
	END_IF
END_FOR

// Should return above if successful
Trace(CONCAT('Part OID not found on track!  (Track: ', CONCAT(Name, ')')));
_Error := TRUE;
END_METHOD

PROPERTY IsClosed : BOOL
GET
IF ipTrack <> 0 THEN
	IsClosed := ipTrack.GetIsClosed();
ELSE
	Trace('IsClosed called before initialization!');
	_Error := TRUE;
END_IF
END_GET
END_PROPERTY

PROPERTY Length : LREAL
GET
IF ipTrack <> 0 THEN
	Length := ipTrack.GetLength();
ELSE
	Trace('Length called before initialization!');
	_Error := TRUE;
END_IF
END_GET
END_PROPERTY

PROPERTY Name : STRING
GET
IF ipTrack <> 0 THEN
	Name := ipTrack.GetObjectName();
ELSE
	Trace('Name called before initialization!');
	_Error := TRUE;
END_IF
END_GET
END_PROPERTY

METHOD PRIVATE Initialize : BOOL
CASE InitializeState OF
	E_InitializeState_Track.eInitializeStateTrack_Check:
		IF ipTrack <> 0 THEN
			InitializeState := E_InitializeState_Track.eInitializeStateTrack_GetPartInfo;
		ELSE
			IF Parameters_XTS.ENABLE_DEBUG_TRACING THEN
				Trace('Track initialization attempted with null reference');
			END_IF

			InitializeState := E_InitializeState_Track.eInitializeStateTrack_Failed;
		END_IF

	E_InitializeState_Track.eInitializeStateTrack_GetPartInfo:
		NumberOfParts := ipTrack.GetPartCount();
		Parts		  REF= ipTrack.GetPartInfoItems();
		IF NumberOfParts = 0 THEN
			IF Parameters_XTS.ENABLE_DEBUG_TRACING THEN
				Trace('No parts associated with this track');
			END_IF

			InitializeState := E_InitializeState_Track.eInitializeStateTrack_Failed;
		ELSE
			InitializeState := E_InitializeState_Track.eInitializeStateTrack_Complete;
		END_IF

	E_InitializeState_Track.eInitializeStateTrack_Complete:
		_Busy	   := FALSE;
		Initialize := TRUE;

	E_InitializeState_Track.eInitializeStateTrack_Failed:
		_Busy  := FALSE;
		_Error := TRUE;
END_CASE
END_METHOD

END_FUNCTION_BLOCK

// Utilities/FB_TrackingRegister_Stations
FUNCTION_BLOCK FB_TrackingRegister_Stations
VAR
	Status			 : ARRAY[1..TcIoXtsEnvironmentParameterList.MaxXtsInfoStation] OF BOOL;
	_StationsToTrack : REFERENCE TO UDINT;
END_VAR

//This FB is just for ease of tracking what group commands have actually completed

METHOD Check : BOOL
VAR_INPUT
	i : UDINT;
END_VAR
IF __ISVALIDREF(_StationsToTrack) THEN
	IF (i >= 1) AND (i <= _StationsToTrack) THEN
		Check := Status[i];
	END_IF
END_IF
END_METHOD

